LIN {X 0,Y 573.243,Z 513.073,A -85,B 0,C 180,E1 -2300.392,E2 -2300.392} C_VEL
LIN {X 0,Y 573.249,Z 513.077,A -85,B 0,C 180,E1 -2303.077,E2 -2303.077} C_VEL
LIN {X 0,Y 573.268,Z 513.077,A -85,B 0,C 180,E1 -2305.671,E2 -2305.671} C_VEL
LIN {X 0,Y 573.242,Z 513.074,A -85,B 0,C 180,E1 -2308.184,E2 -2308.184} C_VEL
LIN {X 0,Y 573.262,Z 513.071,A -85,B 0,C 180,E1 -2310.634,E2 -2310.634} C_VEL
LIN {X 0,Y 573.262,Z 513.081,A -85,B 0,C 180,E1 -2313.499,E2 -2313.499} C_VEL
LIN {X 0,Y 573.224,Z 513.076,A -85,B 0,C 180,E1 -2316.134,E2 -2316.134} C_VEL
LIN {X 0,Y 573.253,Z 513.078,A -85,B 0,C 180,E1 -2319.173,E2 -2319.173} C_VEL
LIN {X 0,Y 573.231,Z 513.084,A -85,B 0,C 180,E1 -2321.411,E2 -2321.411} C_VEL
LIN {X 0,Y 573.249,Z 513.079,A -85,B 0,C 180,E1 -2323.621,E2 -2323.621} C_VEL
LIN {X 0,Y 573.227,Z 513.076,A -85,B 0,C 180,E1 -2326.529,E2 -2326.529} C_VEL
LIN {X 0,Y 573.273,Z 513.07,A -85,B 0,C 180,E1 -2328.733,E2 -2328.733} C_VEL
LIN {X 0,Y 573.298,Z 513.075,A -85,B 0,C 180,E1 -2331.54,E2 -2331.54} C_VEL
LIN {X 0,Y 573.284,Z 513.068,A -85,B 0,C 180,E1 -2334.371,E2 -2334.371} C_VEL
LIN {X 0,Y 573.3,Z 513.069,A -85,B 0,C 180,E1 -2337.892,E2 -2337.892} C_VEL
LIN {X 0,Y 573.328,Z 513.064,A -85,B 0,C 180,E1 -2340.702,E2 -2340.702} C_VEL
LIN {X 0,Y 573.234,Z 513.083,A -85,B 0,C 180,E1 -2343.514,E2 -2343.514} C_VEL
LIN {X 0,Y 573.283,Z 513.075,A -85,B 0,C 180,E1 -2345.628,E2 -2345.628} C_VEL
LIN {X 0,Y 573.298,Z 513.067,A -85,B 0,C 180,E1 -2348.459,E2 -2348.459} C_VEL
LIN {X 0,Y 573.287,Z 513.077,A -85,B 0,C 180,E1 -2351.311,E2 -2351.311} C_VEL
LIN {X 0,Y 573.269,Z 513.071,A -85,B 0,C 180,E1 -2354.425,E2 -2354.425} C_VEL
LIN {X 0,Y 573.249,Z 513.079,A -85,B 0,C 180,E1 -2357.111,E2 -2357.111} C_VEL
LIN {X 0,Y 573.247,Z 513.075,A -85,B 0,C 180,E1 -2360.076,E2 -2360.076} C_VEL
LIN {X 0,Y 573.229,Z 513.076,A -85,B 0,C 180,E1 -2362.338,E2 -2362.338} C_VEL
LIN {X 0,Y 573.24,Z 513.075,A -85,B 0,C 180,E1 -2364.401,E2 -2364.401} C_VEL
LIN {X 0,Y 572.615,Z 513.157,A -85,B 0,C 180,E1 -2364.987,E2 -2364.987} C_VEL
LIN {X 0,Y 569.777,Z 513.516,A -85,B 0,C 180,E1 -2365.939,E2 -2365.939} C_VEL
LIN {X 0,Y 567.349,Z 513.821,A -85,B 0,C 180,E1 -2366.705,E2 -2366.705} C_VEL
LIN {X 0,Y 566.296,Z 513.949,A -85,B 0,C 180,E1 -2367.296,E2 -2367.296} C_VEL
LIN {X 0,Y 566.207,Z 513.958,A -85,B 0,C 180,E1 -2367.496,E2 -2367.496} C_VEL
LIN {X 0,Y 566.246,Z 514.057,A -85,B 0,C 180,E1 -2370.176,E2 -2370.176} C_VEL
LIN {X 0,Y 566.585,Z 517.753,A -85,B 0,C 180,E1 -2370.853,E2 -2370.853} C_VEL
LIN {X 0,Y 566.382,Z 534.137,A -85,B 0,C 180,E1 -2373.762,E2 -2373.762} C_VEL
LIN {X 0,Y 566.229,Z 547.137,A -85,B 0,C 180,E1 -2376.042,E2 -2376.042} C_VEL
LIN {X 0,Y 567.189,Z 554.187,A -85,B 0,C 180,E1 -2376.165,E2 -2376.165} C_VEL
LIN {X 0,Y 566.935,Z 654.262,A -85,B 0,C 180,E1 -2377.453,E2 -2377.453} C_VEL
LIN {X 0,Y 566.822,Z 667.928,A -85,B 0,C 180,E1 -2377.785,E2 -2377.785} C_VEL
LIN {X 0,Y 566.718,Z 679.77,A -85,B 0,C 180,E1 -2378.209,E2 -2378.209} C_VEL
LIN {X 0,Y 566.6,Z 691.935,A -85,B 0,C 180,E1 -2378.797,E2 -2378.797} C_VEL
LIN {X 0,Y 566.436,Z 702.934,A -85,B 0,C 180,E1 -2379.48,E2 -2379.48} C_VEL
LIN {X 0,Y 566.311,Z 713.502,A -85,B 0,C 180,E1 -2380.301,E2 -2380.301} C_VEL
LIN {X 0,Y 566.196,Z 723.392,A -85,B 0,C 180,E1 -2381.255,E2 -2381.255} C_VEL
LIN {X 0,Y 566.063,Z 732.117,A -85,B 0,C 180,E1 -2382.297,E2 -2382.297} C_VEL
LIN {X 0,Y 565.987,Z 738.863,A -85,B 0,C 180,E1 -2383.288,E2 -2383.288} C_VEL
LIN {X 0,Y 565.955,Z 745.455,A -85,B 0,C 180,E1 -2384.502,E2 -2384.502} C_VEL
LIN {X 0,Y 565.911,Z 749.683,A -85,B 0,C 180,E1 -2385.495,E2 -2385.495} C_VEL
LIN {X 0,Y 565.888,Z 753.006,A -85,B 0,C 180,E1 -2386.5,E2 -2386.5} C_VEL
LIN {X 0,Y 565.861,Z 756.162,A -85,B 0,C 180,E1 -2387.882,E2 -2387.882} C_VEL
LIN {X 0,Y 565.825,Z 757.735,A -85,B 0,C 180,E1 -2389.258,E2 -2389.258} C_VEL
LIN {X 0,Y 565.812,Z 757.824,A -85,B 0,C 180,E1 -2390.695,E2 -2390.695} C_VEL
LIN {X 0,Y 565.827,Z 757.03,A -85,B 0,C 180,E1 -2391.61,E2 -2391.61} C_VEL
LIN {X 0,Y 565.843,Z 755.324,A -85,B 0,C 180,E1 -2392.646,E2 -2392.646} C_VEL
LIN {X 0,Y 565.912,Z 752.312,A -85,B 0,C 180,E1 -2393.825,E2 -2393.825} C_VEL
LIN {X 0,Y 565.9,Z 747.388,A -85,B 0,C 180,E1 -2395.162,E2 -2395.162} C_VEL
LIN {X 0,Y 565.984,Z 741.795,A -85,B 0,C 180,E1 -2396.3,E2 -2396.3} C_VEL
LIN {X 0,Y 566.048,Z 734.523,A -85,B 0,C 180,E1 -2397.462,E2 -2397.462} C_VEL
LIN {X 0,Y 566.173,Z 725.725,A -85,B 0,C 180,E1 -2398.578,E2 -2398.578} C_VEL
LIN {X 0,Y 566.257,Z 716.551,A -85,B 0,C 180,E1 -2399.516,E2 -2399.516} C_VEL
LIN {X 0,Y 566.398,Z 706.371,A -85,B 0,C 180,E1 -2400.362,E2 -2400.362} C_VEL
LIN {X 0,Y 566.515,Z 695.904,A -85,B 0,C 180,E1 -2401.066,E2 -2401.066} C_VEL
LIN {X 0,Y 566.678,Z 683.715,A -85,B 0,C 180,E1 -2401.708,E2 -2401.708} C_VEL
LIN {X 0,Y 566.802,Z 671.491,A -85,B 0,C 180,E1 -2402.192,E2 -2402.192} C_VEL
LIN {X 0,Y 566.923,Z 658.595,A -85,B 0,C 180,E1 -2402.549,E2 -2402.549} C_VEL
LIN {X 0,Y 567.017,Z 643.292,A -85,B 0,C 180,E1 -2402.793,E2 -2402.793} C_VEL
LIN {X 0,Y 567.092,Z 552.392,A -85,B 0,C 180,E1 -2403.95,E2 -2403.95} C_VEL
LIN {X 0,Y 566.244,Z 547.089,A -85,B 0,C 180,E1 -2404.056,E2 -2404.056} C_VEL
LIN {X 0,Y 566.406,Z 531.183,A -85,B 0,C 180,E1 -2406.849,E2 -2406.849} C_VEL
LIN {X 0,Y 566.53,Z 516.374,A -85,B 0,C 180,E1 -2409.486,E2 -2409.486} C_VEL
LIN {X 0,Y 566.234,Z 513.954,A -85,B 0,C 180,E1 -2409.949,E2 -2409.949} C_VEL
LIN {X 0,Y 566.22,Z 513.957,A -85,B 0,C 180,E1 -2412.887,E2 -2412.887} C_VEL
LIN {X 0,Y 566.23,Z 513.948,A -85,B 0,C 180,E1 -2415.628,E2 -2415.628} C_VEL
LIN {X 0,Y 566.23,Z 513.955,A -85,B 0,C 180,E1 -2418.676,E2 -2418.676} C_VEL
LIN {X 0,Y 566.226,Z 513.949,A -85,B 0,C 180,E1 -2421.435,E2 -2421.435} C_VEL
LIN {X 0,Y 566.263,Z 513.945,A -85,B 0,C 180,E1 -2424.303,E2 -2424.303} C_VEL
LIN {X 0,Y 566.282,Z 513.94,A -85,B 0,C 180,E1 -2427.867,E2 -2427.867} C_VEL
LIN {X 0,Y 566.301,Z 513.944,A -85,B 0,C 180,E1 -2430.712,E2 -2430.712} C_VEL
LIN {X 0,Y 566.27,Z 513.95,A -85,B 0,C 180,E1 -2432.847,E2 -2432.847} C_VEL
LIN {X 0,Y 566.261,Z 513.944,A -85,B 0,C 180,E1 -2435.699,E2 -2435.699} C_VEL
LIN {X 0,Y 566.226,Z 513.951,A -85,B 0,C 180,E1 -2438.567,E2 -2438.567} C_VEL
LIN {X 0,Y 566.241,Z 513.949,A -85,B 0,C 180,E1 -2441.455,E2 -2441.455} C_VEL
LIN {X 0,Y 566.234,Z 513.948,A -85,B 0,C 180,E1 -2444.508,E2 -2444.508} C_VEL
LIN {X 0,Y 566.199,Z 513.957,A -85,B 0,C 180,E1 -2447.333,E2 -2447.333} C_VEL
LIN {X 0,Y 566.213,Z 513.949,A -85,B 0,C 180,E1 -2450.338,E2 -2450.338} C_VEL
LIN {X 0,Y 566.17,Z 513.962,A -85,B 0,C 180,E1 -2453.282,E2 -2453.282} C_VEL
LIN {X 0,Y 566.213,Z 513.951,A -85,B 0,C 180,E1 -2455.75,E2 -2455.75} C_VEL
LIN {X 0,Y 566.203,Z 513.95,A -85,B 0,C 180,E1 -2458.203,E2 -2458.203} C_VEL
LIN {X 0,Y 566.201,Z 513.958,A -85,B 0,C 180,E1 -2461.079,E2 -2461.079} C_VEL
LIN {X 0,Y 566.213,Z 513.952,A -85,B 0,C 180,E1 -2463.735,E2 -2463.735} C_VEL
LIN {X 0,Y 566.201,Z 513.951,A -85,B 0,C 180,E1 -2466.571,E2 -2466.571} C_VEL
LIN {X 0,Y 566.223,Z 513.958,A -85,B 0,C 180,E1 -2469.274,E2 -2469.274} C_VEL
LIN {X 0,Y 566.217,Z 513.949,A -85,B 0,C 180,E1 -2472.088,E2 -2472.088} C_VEL
LIN {X 0,Y 566.176,Z 513.958,A -85,B 0,C 180,E1 -2475.037,E2 -2475.037} C_VEL
LIN {X 0,Y 566.191,Z 513.954,A -85,B 0,C 180,E1 -2477.911,E2 -2477.911} C_VEL
LIN {X 0,Y 566.224,Z 513.948,A -85,B 0,C 180,E1 -2480.728,E2 -2480.728} C_VEL
LIN {X 0,Y 566.188,Z 513.957,A -85,B 0,C 180,E1 -2483.789,E2 -2483.789} C_VEL
LIN {X 0,Y 566.216,Z 513.949,A -85,B 0,C 180,E1 -2486.266,E2 -2486.266} C_VEL
LIN {X 0,Y 566.194,Z 513.953,A -85,B 0,C 180,E1 -2488.924,E2 -2488.924} C_VEL
LIN {X 0,Y 566.216,Z 513.954,A -85,B 0,C 180,E1 -2491.858,E2 -2491.858} C_VEL
LIN {X 0,Y 566.219,Z 513.949,A -85,B 0,C 180,E1 -2494.252,E2 -2494.252} C_VEL
LIN {X 0,Y 566.174,Z 513.954,A -85,B 0,C 180,E1 -2496.72,E2 -2496.72} C_VEL
LIN {X 0,Y 566.212,Z 513.959,A -85,B 0,C 180,E1 -2499.663,E2 -2499.663} C_VEL
LIN {X 0,Y 566.205,Z 513.95,A -85,B 0,C 180,E1 -2502.669,E2 -2502.669} C_VEL
LIN {X 0,Y 566.239,Z 513.955,A -85,B 0,C 180,E1 -2505.627,E2 -2505.627} C_VEL
LIN {X 0,Y 566.241,Z 513.945,A -85,B 0,C 180,E1 -2508.676,E2 -2508.676} C_VEL
LIN {X 0,Y 566.233,Z 513.952,A -85,B 0,C 180,E1 -2511.435,E2 -2511.435} C_VEL
LIN {X 0,Y 566.261,Z 513.945,A -85,B 0,C 180,E1 -2514.302,E2 -2514.302} C_VEL
LIN {X 0,Y 566.285,Z 513.949,A -85,B 0,C 180,E1 -2517.867,E2 -2517.867} C_VEL
LIN {X 0,Y 566.307,Z 513.937,A -85,B 0,C 180,E1 -2520.711,E2 -2520.711} C_VEL
LIN {X 0,Y 566.278,Z 513.941,A -85,B 0,C 180,E1 -2522.846,E2 -2522.846} C_VEL
LIN {X 0,Y 566.264,Z 513.95,A -85,B 0,C 180,E1 -2525.699,E2 -2525.699} C_VEL
LIN {X 0,Y 566.233,Z 513.948,A -85,B 0,C 180,E1 -2528.566,E2 -2528.566} C_VEL
LIN {X 0,Y 566.249,Z 513.947,A -85,B 0,C 180,E1 -2531.455,E2 -2531.455} C_VEL
LIN {X 0,Y 566.242,Z 513.948,A -85,B 0,C 180,E1 -2534.507,E2 -2534.507} C_VEL
LIN {X 0,Y 566.206,Z 513.951,A -85,B 0,C 180,E1 -2537.332,E2 -2537.332} C_VEL
LIN {X 0,Y 566.215,Z 513.954,A -85,B 0,C 180,E1 -2540.337,E2 -2540.337} C_VEL
LIN {X 0,Y 566.177,Z 513.954,A -85,B 0,C 180,E1 -2543.281,E2 -2543.281} C_VEL
LIN {X 0,Y 566.22,Z 513.953,A -85,B 0,C 180,E1 -2545.749,E2 -2545.749} C_VEL
LIN {X 0,Y 566.21,Z 513.958,A -85,B 0,C 180,E1 -2548.202,E2 -2548.202} C_VEL
LIN {X 0,Y 566.197,Z 513.951,A -85,B 0,C 180,E1 -2551.076,E2 -2551.076} C_VEL
LIN {X 0,Y 566.205,Z 513.953,A -85,B 0,C 180,E1 -2553.732,E2 -2553.732} C_VEL
LIN {X 0,Y 566.215,Z 513.953,A -85,B 0,C 180,E1 -2556.569,E2 -2556.569} C_VEL
LIN {X 0,Y 566.222,Z 513.95,A -85,B 0,C 180,E1 -2559.686,E2 -2559.686} C_VEL
LIN {X 0,Y 566.2,Z 513.952,A -85,B 0,C 180,E1 -2562.916,E2 -2562.916} C_VEL
LIN {X 0,Y 566.206,Z 513.956,A -85,B 0,C 180,E1 -2566.048,E2 -2566.048} C_VEL
LIN {X 0,Y 566.211,Z 513.949,A -85,B 0,C 180,E1 -2569.214,E2 -2569.214} C_VEL
LIN {X 0,Y 566.19,Z 513.953,A -85,B 0,C 180,E1 -2571.636,E2 -2571.636} C_VEL
LIN {X 0,Y 566.169,Z 513.964,A -85,B 0,C 180,E1 -2574.307,E2 -2574.307} C_VEL
LIN {X 0,Y 566.227,Z 513.95,A -85,B 0,C 180,E1 -2576.897,E2 -2576.897} C_VEL
LIN {X 0,Y 566.187,Z 513.953,A -85,B 0,C 180,E1 -2579.407,E2 -2579.407} C_VEL
LIN {X 0,Y 566.219,Z 513.95,A -85,B 0,C 180,E1 -2581.857,E2 -2581.857} C_VEL
LIN {X 0,Y 566.216,Z 513.956,A -85,B 0,C 180,E1 -2584.25,E2 -2584.25} C_VEL
LIN {X 0,Y 566.187,Z 514.013,A -85,B 0,C 180,E1 -2586.754,E2 -2586.754} C_VEL
LIN {X 0,Y 567.076,Z 519.274,A -85,B 0,C 180,E1 -2587.597,E2 -2587.597} C_VEL
LIN {X 0,Y 566.791,Z 539.041,A -85,B 0,C 180,E1 -2590.571,E2 -2590.571} C_VEL
LIN {X 0,Y 566.558,Z 557.196,A -85,B 0,C 180,E1 -2593.257,E2 -2593.257} C_VEL
LIN {X 0,Y 566.399,Z 576.069,A -85,B 0,C 180,E1 -2595.997,E2 -2595.997} C_VEL
LIN {X 0,Y 567.211,Z 583.224,A -85,B 0,C 180,E1 -2596.109,E2 -2596.109} C_VEL
LIN {X 0,Y 566.94,Z 683.899,A -85,B 0,C 180,E1 -2597.402,E2 -2597.402} C_VEL
LIN {X 0,Y 566.837,Z 697.187,A -85,B 0,C 180,E1 -2597.718,E2 -2597.718} C_VEL
LIN {X 0,Y 566.758,Z 709.351,A -85,B 0,C 180,E1 -2598.148,E2 -2598.148} C_VEL
LIN {X 0,Y 566.606,Z 721.341,A -85,B 0,C 180,E1 -2598.718,E2 -2598.718} C_VEL
LIN {X 0,Y 566.461,Z 733.188,A -85,B 0,C 180,E1 -2599.454,E2 -2599.454} C_VEL
LIN {X 0,Y 566.319,Z 743.59,A -85,B 0,C 180,E1 -2600.264,E2 -2600.264} C_VEL
LIN {X 0,Y 566.207,Z 752.103,A -85,B 0,C 180,E1 -2601.073,E2 -2601.073} C_VEL
LIN {X 0,Y 566.113,Z 759.953,A -85,B 0,C 180,E1 -2601.971,E2 -2601.971} C_VEL
LIN {X 0,Y 566.005,Z 767.615,A -85,B 0,C 180,E1 -2603.046,E2 -2603.046} C_VEL
LIN {X 0,Y 566.004,Z 774.675,A -85,B 0,C 180,E1 -2604.298,E2 -2604.298} C_VEL
LIN {X 0,Y 565.933,Z 779.368,A -85,B 0,C 180,E1 -2605.369,E2 -2605.369} C_VEL
LIN {X 0,Y 565.927,Z 782.954,A -85,B 0,C 180,E1 -2606.439,E2 -2606.439} C_VEL
LIN {X 0,Y 565.878,Z 784.806,A -85,B 0,C 180,E1 -2607.151,E2 -2607.151} C_VEL
LIN {X 0,Y 565.846,Z 787.185,A -85,B 0,C 180,E1 -2608.576,E2 -2608.576} C_VEL
LIN {X 0,Y 565.839,Z 788,A -85,B 0,C 180,E1 -2609.999,E2 -2609.999} C_VEL
LIN {X 0,Y 565.846,Z 787.188,A -85,B 0,C 180,E1 -2611.422,E2 -2611.422} C_VEL
LIN {X 0,Y 565.878,Z 784.812,A -85,B 0,C 180,E1 -2612.847,E2 -2612.847} C_VEL
LIN {X 0,Y 565.926,Z 781.899,A -85,B 0,C 180,E1 -2613.915,E2 -2613.915} C_VEL
LIN {X 0,Y 565.878,Z 777.953,A -85,B 0,C 180,E1 -2614.986,E2 -2614.986} C_VEL
LIN {X 0,Y 566.001,Z 772.872,A -85,B 0,C 180,E1 -2616.057,E2 -2616.057} C_VEL
LIN {X 0,Y 566.04,Z 766.476,A -85,B 0,C 180,E1 -2617.131,E2 -2617.131} C_VEL
LIN {X 0,Y 566.133,Z 758.487,A -85,B 0,C 180,E1 -2618.207,E2 -2618.207} C_VEL
LIN {X 0,Y 566.228,Z 750.347,A -85,B 0,C 180,E1 -2619.104,E2 -2619.104} C_VEL
LIN {X 0,Y 566.34,Z 740.414,A -85,B 0,C 180,E1 -2620.004,E2 -2620.004} C_VEL
LIN {X 0,Y 566.514,Z 729.301,A -85,B 0,C 180,E1 -2620.807,E2 -2620.807} C_VEL
LIN {X 0,Y 566.659,Z 718.199,A -85,B 0,C 180,E1 -2621.445,E2 -2621.445} C_VEL
LIN {X 0,Y 566.738,Z 706.012,A -85,B 0,C 180,E1 -2621.987,E2 -2621.987} C_VEL
LIN {X 0,Y 566.911,Z 693.222,A -85,B 0,C 180,E1 -2622.392,E2 -2622.392} C_VEL
LIN {X 0,Y 566.981,Z 681.182,A -85,B 0,C 180,E1 -2622.641,E2 -2622.641} C_VEL
LIN {X 0,Y 567.029,Z 580.268,A -85,B 0,C 180,E1 -2623.934,E2 -2623.934} C_VEL
LIN {X 0,Y 566.389,Z 575.8,A -85,B 0,C 180,E1 -2624.024,E2 -2624.024} C_VEL
LIN {X 0,Y 566.587,Z 554.721,A -85,B 0,C 180,E1 -2627.107,E2 -2627.107} C_VEL
LIN {X 0,Y 566.849,Z 534.4,A -85,B 0,C 180,E1 -2630.123,E2 -2630.123} C_VEL
LIN {X 0,Y 567.093,Z 519.288,A -85,B 0,C 180,E1 -2632.4,E2 -2632.4} C_VEL
LIN {X 0,Y 566.188,Z 513.964,A -85,B 0,C 180,E1 -2633.284,E2 -2633.284} C_VEL
LIN {X 0,Y 566.212,Z 513.957,A -85,B 0,C 180,E1 -2635.748,E2 -2635.748} C_VEL
LIN {X 0,Y 566.2,Z 513.954,A -85,B 0,C 180,E1 -2638.201,E2 -2638.201} C_VEL
LIN {X 0,Y 566.197,Z 513.957,A -85,B 0,C 180,E1 -2641.077,E2 -2641.077} C_VEL
LIN {X 0,Y 566.208,Z 513.956,A -85,B 0,C 180,E1 -2643.733,E2 -2643.733} C_VEL
LIN {X 0,Y 566.207,Z 513.951,A -85,B 0,C 180,E1 -2646.568,E2 -2646.568} C_VEL
LIN {X 0,Y 566.208,Z 513.957,A -85,B 0,C 180,E1 -2649.684,E2 -2649.684} C_VEL
LIN {X 0,Y 566.21,Z 513.952,A -85,B 0,C 180,E1 -2652.086,E2 -2652.086} C_VEL
LIN {X 0,Y 566.167,Z 513.959,A -85,B 0,C 180,E1 -2655.035,E2 -2655.035} C_VEL
LIN {X 0,Y 566.211,Z 513.951,A -85,B 0,C 180,E1 -2658.135,E2 -2658.135} C_VEL
LIN {X 0,Y 566.216,Z 513.95,A -85,B 0,C 180,E1 -2660.726,E2 -2660.726} C_VEL
LIN {X 0,Y 566.211,Z 513.954,A -85,B 0,C 180,E1 -2663.782,E2 -2663.782} C_VEL
LIN {X 0,Y 566.222,Z 513.948,A -85,B 0,C 180,E1 -2666.262,E2 -2666.262} C_VEL
LIN {X 0,Y 566.194,Z 513.954,A -85,B 0,C 180,E1 -2668.92,E2 -2668.92} C_VEL
LIN {X 0,Y 566.189,Z 513.956,A -85,B 0,C 180,E1 -2671.046,E2 -2671.046} C_VEL
LIN {X 0,Y 566.237,Z 513.956,A -85,B 0,C 180,E1 -2673.46,E2 -2673.46} C_VEL
LIN {X 0,Y 566.19,Z 513.955,A -85,B 0,C 180,E1 -2675.819,E2 -2675.819} C_VEL
LIN {X 0,Y 566.208,Z 513.952,A -85,B 0,C 180,E1 -2678.902,E2 -2678.902} C_VEL
LIN {X 0,Y 566.205,Z 513.955,A -85,B 0,C 180,E1 -2681.172,E2 -2681.172} C_VEL
LIN {X 0,Y 566.211,Z 513.959,A -85,B 0,C 180,E1 -2683.412,E2 -2683.412} C_VEL
LIN {X 0,Y 566.19,Z 513.952,A -85,B 0,C 180,E1 -2686.358,E2 -2686.358} C_VEL
LIN {X 0,Y 566.265,Z 513.942,A -85,B 0,C 180,E1 -2688.653,E2 -2688.653} C_VEL
LIN {X 0,Y 566.239,Z 513.955,A -85,B 0,C 180,E1 -2691.434,E2 -2691.434} C_VEL
LIN {X 0,Y 566.251,Z 513.945,A -85,B 0,C 180,E1 -2694.301,E2 -2694.301} C_VEL
LIN {X 0,Y 566.271,Z 513.945,A -85,B 0,C 180,E1 -2697.866,E2 -2697.866} C_VEL
LIN {X 0,Y 566.298,Z 513.94,A -85,B 0,C 180,E1 -2700.711,E2 -2700.711} C_VEL
LIN {X 0,Y 566.27,Z 513.944,A -85,B 0,C 180,E1 -2702.845,E2 -2702.845} C_VEL
LIN {X 0,Y 566.251,Z 513.95,A -85,B 0,C 180,E1 -2705.698,E2 -2705.698} C_VEL
LIN {X 0,Y 566.239,Z 513.947,A -85,B 0,C 180,E1 -2708.565,E2 -2708.565} C_VEL
LIN {X 0,Y 566.239,Z 513.956,A -85,B 0,C 180,E1 -2711.454,E2 -2711.454} C_VEL
LIN {X 0,Y 566.222,Z 513.949,A -85,B 0,C 180,E1 -2714.507,E2 -2714.507} C_VEL
LIN {X 0,Y 566.194,Z 513.962,A -85,B 0,C 180,E1 -2717.331,E2 -2717.331} C_VEL
LIN {X 0,Y 566.209,Z 513.95,A -85,B 0,C 180,E1 -2720.337,E2 -2720.337} C_VEL
LIN {X 0,Y 566.179,Z 513.963,A -85,B 0,C 180,E1 -2723.404,E2 -2723.404} C_VEL
LIN {X 0,Y 566.216,Z 513.955,A -85,B 0,C 180,E1 -2725.748,E2 -2725.748} C_VEL
LIN {X 0,Y 566.207,Z 513.958,A -85,B 0,C 180,E1 -2727.496,E2 -2727.496} C_VEL
LIN {X 0,Y 565.52,Z 514.041,A -85,B 0,C 180,E1 -2727.892,E2 -2727.892} C_VEL
LIN {X 0,Y 559.819,Z 514.755,A -85,B 0,C 180,E1 -2729.137,E2 -2729.137} C_VEL
LIN {X 0,Y 559.155,Z 514.837,A -85,B 0,C 180,E1 -2729.54,E2 -2729.54} C_VEL
LIN {X 0,Y 559.213,Z 514.972,A -85,B 0,C 180,E1 -2730.083,E2 -2730.083} C_VEL
LIN {X 0,Y 559.566,Z 519.903,A -85,B 0,C 180,E1 -2730.994,E2 -2730.994} C_VEL
LIN {X 0,Y 559.377,Z 535.33,A -85,B 0,C 180,E1 -2733.766,E2 -2733.766} C_VEL
LIN {X 0,Y 559.188,Z 547.236,A -85,B 0,C 180,E1 -2735.873,E2 -2735.873} C_VEL
LIN {X 0,Y 560.272,Z 553.876,A -85,B 0,C 180,E1 -2735.987,E2 -2735.987} C_VEL
LIN {X 0,Y 560.022,Z 654.191,A -85,B 0,C 180,E1 -2737.293,E2 -2737.293} C_VEL
LIN {X 0,Y 559.9,Z 667.815,A -85,B 0,C 180,E1 -2737.627,E2 -2737.627} C_VEL
LIN {X 0,Y 559.755,Z 680.312,A -85,B 0,C 180,E1 -2738.081,E2 -2738.081} C_VEL
LIN {X 0,Y 559.621,Z 692.123,A -85,B 0,C 180,E1 -2738.666,E2 -2738.666} C_VEL
LIN {X 0,Y 559.433,Z 703.358,A -85,B 0,C 180,E1 -2739.376,E2 -2739.376} C_VEL
LIN {X 0,Y 559.296,Z 714.193,A -85,B 0,C 180,E1 -2740.239,E2 -2740.239} C_VEL
LIN {X 0,Y 559.136,Z 723.82,A -85,B 0,C 180,E1 -2741.19,E2 -2741.19} C_VEL
LIN {X 0,Y 559.007,Z 732.434,A -85,B 0,C 180,E1 -2742.241,E2 -2742.241} C_VEL
LIN {X 0,Y 558.896,Z 740.27,A -85,B 0,C 180,E1 -2743.44,E2 -2743.44} C_VEL
LIN {X 0,Y 558.863,Z 745.614,A -85,B 0,C 180,E1 -2744.465,E2 -2744.465} C_VEL
LIN {X 0,Y 558.814,Z 750.957,A -85,B 0,C 180,E1 -2745.796,E2 -2745.796} C_VEL
LIN {X 0,Y 558.759,Z 754.941,A -85,B 0,C 180,E1 -2747.22,E2 -2747.22} C_VEL
LIN {X 0,Y 558.756,Z 756.676,A -85,B 0,C 180,E1 -2748.194,E2 -2748.194} C_VEL
LIN {X 0,Y 558.742,Z 757.674,A -85,B 0,C 180,E1 -2749.153,E2 -2749.153} C_VEL
LIN {X 0,Y 558.753,Z 757.993,A -85,B 0,C 180,E1 -2750.108,E2 -2750.108} C_VEL
LIN {X 0,Y 558.724,Z 757.44,A -85,B 0,C 180,E1 -2751.249,E2 -2751.249} C_VEL
LIN {X 0,Y 558.744,Z 755.844,A -85,B 0,C 180,E1 -2752.412,E2 -2752.412} C_VEL
LIN {X 0,Y 558.835,Z 752.621,A -85,B 0,C 180,E1 -2753.768,E2 -2753.768} C_VEL
LIN {X 0,Y 558.804,Z 748.993,A -85,B 0,C 180,E1 -2754.834,E2 -2754.834} C_VEL
LIN {X 0,Y 558.871,Z 743.311,A -85,B 0,C 180,E1 -2756.095,E2 -2756.095} C_VEL
LIN {X 0,Y 558.948,Z 736.432,A -85,B 0,C 180,E1 -2757.273,E2 -2757.273} C_VEL
LIN {X 0,Y 559.049,Z 729.01,A -85,B 0,C 180,E1 -2758.295,E2 -2758.295} C_VEL
LIN {X 0,Y 559.193,Z 720.027,A -85,B 0,C 180,E1 -2759.299,E2 -2759.299} C_VEL
LIN {X 0,Y 559.329,Z 710.35,A -85,B 0,C 180,E1 -2760.179,E2 -2760.179} C_VEL
LIN {X 0,Y 559.475,Z 699.524,A -85,B 0,C 180,E1 -2760.976,E2 -2760.976} C_VEL
LIN {X 0,Y 559.644,Z 688.739,A -85,B 0,C 180,E1 -2761.608,E2 -2761.608} C_VEL
LIN {X 0,Y 559.827,Z 676.28,A -85,B 0,C 180,E1 -2762.172,E2 -2762.172} C_VEL
LIN {X 0,Y 559.943,Z 663.4,A -85,B 0,C 180,E1 -2762.589,E2 -2762.589} C_VEL
LIN {X 0,Y 560.047,Z 650.613,A -85,B 0,C 180,E1 -2762.853,E2 -2762.853} C_VEL
LIN {X 0,Y 560.246,Z 553.607,A -85,B 0,C 180,E1 -2764.108,E2 -2764.108} C_VEL
LIN {X 0,Y 559.228,Z 547.111,A -85,B 0,C 180,E1 -2764.232,E2 -2764.232} C_VEL
LIN {X 0,Y 559.468,Z 529.99,A -85,B 0,C 180,E1 -2767.278,E2 -2767.278} C_VEL
LIN {X 0,Y 559.506,Z 517.138,A -85,B 0,C 180,E1 -2769.601,E2 -2769.601} C_VEL
LIN {X 0,Y 559.197,Z 514.831,A -85,B 0,C 180,E1 -2770.069,E2 -2770.069} C_VEL
LIN {X 0,Y 559.178,Z 514.83,A -85,B 0,C 180,E1 -2773.199,E2 -2773.199} C_VEL
LIN {X 0,Y 559.171,Z 514.829,A -85,B 0,C 180,E1 -2776.185,E2 -2776.185} C_VEL
LIN {X 0,Y 559.191,Z 514.828,A -85,B 0,C 180,E1 -2779.135,E2 -2779.135} C_VEL
LIN {X 0,Y 559.203,Z 514.823,A -85,B 0,C 180,E1 -2782.055,E2 -2782.055} C_VEL
LIN {X 0,Y 559.252,Z 514.825,A -85,B 0,C 180,E1 -2784.954,E2 -2784.954} C_VEL
LIN {X 0,Y 559.253,Z 514.816,A -85,B 0,C 180,E1 -2787.84,E2 -2787.84} C_VEL
LIN {X 0,Y 559.271,Z 514.82,A -85,B 0,C 180,E1 -2790.721,E2 -2790.721} C_VEL
LIN {X 0,Y 559.237,Z 514.827,A -85,B 0,C 180,E1 -2792.882,E2 -2792.882} C_VEL
LIN {X 0,Y 559.229,Z 514.819,A -85,B 0,C 180,E1 -2795.771,E2 -2795.771} C_VEL
LIN {X 0,Y 559.185,Z 514.829,A -85,B 0,C 180,E1 -2798.675,E2 -2798.675} C_VEL
LIN {X 0,Y 559.205,Z 514.824,A -85,B 0,C 180,E1 -2801.601,E2 -2801.601} C_VEL
LIN {X 0,Y 559.199,Z 514.825,A -85,B 0,C 180,E1 -2804.596,E2 -2804.596} C_VEL
LIN {X 0,Y 559.142,Z 514.833,A -85,B 0,C 180,E1 -2807.558,E2 -2807.558} C_VEL
LIN {X 0,Y 559.172,Z 514.827,A -85,B 0,C 180,E1 -2809.838,E2 -2809.838} C_VEL
LIN {X 0,Y 559.141,Z 514.83,A -85,B 0,C 180,E1 -2812.154,E2 -2812.154} C_VEL
LIN {X 0,Y 559.176,Z 514.834,A -85,B 0,C 180,E1 -2815.299,E2 -2815.299} C_VEL
LIN {X 0,Y 559.158,Z 514.83,A -85,B 0,C 180,E1 -2817.714,E2 -2817.714} C_VEL
LIN {X 0,Y 559.158,Z 514.828,A -85,B 0,C 180,E1 -2820.183,E2 -2820.183} C_VEL
LIN {X 0,Y 559.159,Z 514.83,A -85,B 0,C 180,E1 -2822.716,E2 -2822.716} C_VEL
LIN {X 0,Y 559.129,Z 514.841,A -85,B 0,C 180,E1 -2825.325,E2 -2825.325} C_VEL
LIN {X 0,Y 559.137,Z 514.831,A -85,B 0,C 180,E1 -2828.018,E2 -2828.018} C_VEL
LIN {X 0,Y 559.193,Z 514.829,A -85,B 0,C 180,E1 -2831.055,E2 -2831.055} C_VEL
LIN {X 0,Y 559.165,Z 514.831,A -85,B 0,C 180,E1 -2833.732,E2 -2833.732} C_VEL
LIN {X 0,Y 559.148,Z 514.831,A -85,B 0,C 180,E1 -2836.804,E2 -2836.804} C_VEL
LIN {X 0,Y 559.176,Z 514.832,A -85,B 0,C 180,E1 -2839.19,E2 -2839.19} C_VEL
LIN {X 0,Y 559.137,Z 514.833,A -85,B 0,C 180,E1 -2841.983,E2 -2841.983} C_VEL
LIN {X 0,Y 559.138,Z 514.831,A -85,B 0,C 180,E1 -2844.787,E2 -2844.787} C_VEL
LIN {X 0,Y 559.177,Z 514.833,A -85,B 0,C 180,E1 -2847.362,E2 -2847.362} C_VEL
LIN {X 0,Y 559.153,Z 514.83,A -85,B 0,C 180,E1 -2850.143,E2 -2850.143} C_VEL
LIN {X 0,Y 559.173,Z 514.829,A -85,B 0,C 180,E1 -2853.098,E2 -2853.098} C_VEL
LIN {X 0,Y 559.161,Z 514.836,A -85,B 0,C 180,E1 -2855.496,E2 -2855.496} C_VEL
LIN {X 0,Y 559.177,Z 514.825,A -85,B 0,C 180,E1 -2858.625,E2 -2858.625} C_VEL
LIN {X 0,Y 559.167,Z 514.827,A -85,B 0,C 180,E1 -2860.927,E2 -2860.927} C_VEL
LIN {X 0,Y 559.171,Z 514.832,A -85,B 0,C 180,E1 -2863.948,E2 -2863.948} C_VEL
LIN {X 0,Y 559.176,Z 514.828,A -85,B 0,C 180,E1 -2866.185,E2 -2866.185} C_VEL
LIN {X 0,Y 559.2,Z 514.824,A -85,B 0,C 180,E1 -2869.134,E2 -2869.134} C_VEL
LIN {X 0,Y 559.209,Z 514.826,A -85,B 0,C 180,E1 -2872.054,E2 -2872.054} C_VEL
LIN {X 0,Y 559.258,Z 514.815,A -85,B 0,C 180,E1 -2874.954,E2 -2874.954} C_VEL
LIN {X 0,Y 559.257,Z 514.825,A -85,B 0,C 180,E1 -2877.84,E2 -2877.84} C_VEL
LIN {X 0,Y 559.278,Z 514.813,A -85,B 0,C 180,E1 -2880.72,E2 -2880.72} C_VEL
LIN {X 0,Y 559.244,Z 514.817,A -85,B 0,C 180,E1 -2882.882,E2 -2882.882} C_VEL
LIN {X 0,Y 559.234,Z 514.827,A -85,B 0,C 180,E1 -2885.77,E2 -2885.77} C_VEL
LIN {X 0,Y 559.192,Z 514.824,A -85,B 0,C 180,E1 -2888.675,E2 -2888.675} C_VEL
LIN {X 0,Y 559.213,Z 514.826,A -85,B 0,C 180,E1 -2891.601,E2 -2891.601} C_VEL
LIN {X 0,Y 559.208,Z 514.823,A -85,B 0,C 180,E1 -2894.596,E2 -2894.596} C_VEL
LIN {X 0,Y 559.149,Z 514.832,A -85,B 0,C 180,E1 -2897.558,E2 -2897.558} C_VEL
LIN {X 0,Y 559.173,Z 514.833,A -85,B 0,C 180,E1 -2899.838,E2 -2899.838} C_VEL
LIN {X 0,Y 559.149,Z 514.838,A -85,B 0,C 180,E1 -2902.153,E2 -2902.153} C_VEL
LIN {X 0,Y 559.184,Z 514.825,A -85,B 0,C 180,E1 -2905.298,E2 -2905.298} C_VEL
LIN {X 0,Y 559.176,Z 514.831,A -85,B 0,C 180,E1 -2908.381,E2 -2908.381} C_VEL
LIN {X 0,Y 559.153,Z 514.828,A -85,B 0,C 180,E1 -2911.273,E2 -2911.273} C_VEL
LIN {X 0,Y 559.164,Z 514.833,A -85,B 0,C 180,E1 -2913.948,E2 -2913.948} C_VEL
LIN {X 0,Y 559.165,Z 514.833,A -85,B 0,C 180,E1 -2916.447,E2 -2916.447} C_VEL
LIN {X 0,Y 559.181,Z 514.826,A -85,B 0,C 180,E1 -2918.934,E2 -2918.934} C_VEL
LIN {X 0,Y 559.169,Z 514.829,A -85,B 0,C 180,E1 -2921.77,E2 -2921.77} C_VEL
LIN {X 0,Y 559.136,Z 514.834,A -85,B 0,C 180,E1 -2924.74,E2 -2924.74} C_VEL
LIN {X 0,Y 559.167,Z 514.827,A -85,B 0,C 180,E1 -2927.256,E2 -2927.256} C_VEL
LIN {X 0,Y 559.186,Z 514.831,A -85,B 0,C 180,E1 -2930.134,E2 -2930.134} C_VEL
LIN {X 0,Y 559.147,Z 514.831,A -85,B 0,C 180,E1 -2932.891,E2 -2932.891} C_VEL
LIN {X 0,Y 559.173,Z 514.83,A -85,B 0,C 180,E1 -2936.05,E2 -2936.05} C_VEL
LIN {X 0,Y 559.162,Z 514.83,A -85,B 0,C 180,E1 -2938.98,E2 -2938.98} C_VEL
LIN {X 0,Y 559.175,Z 514.827,A -85,B 0,C 180,E1 -2941.618,E2 -2941.618} C_VEL
LIN {X 0,Y 559.184,Z 514.828,A -85,B 0,C 180,E1 -2943.902,E2 -2943.902} C_VEL
LIN {X 0,Y 559.165,Z 514.956,A -85,B 0,C 180,E1 -2946.612,E2 -2946.612} C_VEL
LIN {X 0,Y 560.141,Z 520.502,A -85,B 0,C 180,E1 -2947.499,E2 -2947.499} C_VEL
LIN {X 0,Y 559.83,Z 539.763,A -85,B 0,C 180,E1 -2950.429,E2 -2950.429} C_VEL
LIN {X 0,Y 559.589,Z 556.387,A -85,B 0,C 180,E1 -2952.922,E2 -2952.922} C_VEL
LIN {X 0,Y 559.39,Z 576.069,A -85,B 0,C 180,E1 -2955.818,E2 -2955.818} C_VEL
LIN {X 0,Y 560.313,Z 583.224,A -85,B 0,C 180,E1 -2955.934,E2 -2955.934} C_VEL
LIN {X 0,Y 560.02,Z 683.899,A -85,B 0,C 180,E1 -2957.243,E2 -2957.243} C_VEL
LIN {X 0,Y 559.921,Z 697.187,A -85,B 0,C 180,E1 -2957.563,E2 -2957.563} C_VEL
LIN {X 0,Y 559.81,Z 709.353,A -85,B 0,C 180,E1 -2957.998,E2 -2957.998} C_VEL
LIN {X 0,Y 559.631,Z 721.177,A -85,B 0,C 180,E1 -2958.566,E2 -2958.566} C_VEL
LIN {X 0,Y 559.486,Z 733.186,A -85,B 0,C 180,E1 -2959.321,E2 -2959.321} C_VEL
LIN {X 0,Y 559.299,Z 743.591,A -85,B 0,C 180,E1 -2960.141,E2 -2960.141} C_VEL
LIN {X 0,Y 559.162,Z 752.103,A -85,B 0,C 180,E1 -2960.96,E2 -2960.96} C_VEL
LIN {X 0,Y 559.05,Z 759.953,A -85,B 0,C 180,E1 -2961.869,E2 -2961.869} C_VEL
LIN {X 0,Y 558.936,Z 767.727,A -85,B 0,C 180,E1 -2962.975,E2 -2962.975} C_VEL
LIN {X 0,Y 558.936,Z 774.675,A -85,B 0,C 180,E1 -2964.226,E2 -2964.226} C_VEL
LIN {X 0,Y 558.827,Z 779.368,A -85,B 0,C 180,E1 -2965.31,E2 -2965.31} C_VEL
LIN {X 0,Y 558.836,Z 782.955,A -85,B 0,C 180,E1 -2966.394,E2 -2966.394} C_VEL
LIN {X 0,Y 558.799,Z 784.806,A -85,B 0,C 180,E1 -2967.115,E2 -2967.115} C_VEL
LIN {X 0,Y 558.745,Z 787.184,A -85,B 0,C 180,E1 -2968.557,E2 -2968.557} C_VEL
LIN {X 0,Y 558.74,Z 788,A -85,B 0,C 180,E1 -2969.999,E2 -2969.999} C_VEL
LIN {X 0,Y 558.745,Z 787.187,A -85,B 0,C 180,E1 -2971.44,E2 -2971.44} C_VEL
LIN {X 0,Y 558.799,Z 784.812,A -85,B 0,C 180,E1 -2972.883,E2 -2972.883} C_VEL
LIN {X 0,Y 558.843,Z 781.899,A -85,B 0,C 180,E1 -2973.965,E2 -2973.965} C_VEL
LIN {X 0,Y 558.798,Z 777.953,A -85,B 0,C 180,E1 -2975.05,E2 -2975.05} C_VEL
LIN {X 0,Y 558.917,Z 772.872,A -85,B 0,C 180,E1 -2976.134,E2 -2976.134} C_VEL
LIN {X 0,Y 558.977,Z 766.475,A -85,B 0,C 180,E1 -2977.222,E2 -2977.222} C_VEL
LIN {X 0,Y 559.098,Z 758.487,A -85,B 0,C 180,E1 -2978.311,E2 -2978.311} C_VEL
LIN {X 0,Y 559.184,Z 750.346,A -85,B 0,C 180,E1 -2979.22,E2 -2979.22} C_VEL
LIN {X 0,Y 559.352,Z 740.414,A -85,B 0,C 180,E1 -2980.13,E2 -2980.13} C_VEL
LIN {X 0,Y 559.535,Z 729.381,A -85,B 0,C 180,E1 -2980.938,E2 -2980.938} C_VEL
LIN {X 0,Y 559.702,Z 717.164,A -85,B 0,C 180,E1 -2981.643,E2 -2981.643} C_VEL
LIN {X 0,Y 559.819,Z 704.8,A -85,B 0,C 180,E1 -2982.183,E2 -2982.183} C_VEL
LIN {X 0,Y 559.98,Z 691.393,A -85,B 0,C 180,E1 -2982.594,E2 -2982.594} C_VEL
LIN {X 0,Y 560.101,Z 678.165,A -85,B 0,C 180,E1 -2982.845,E2 -2982.845} C_VEL
LIN {X 0,Y 560.2,Z 581.374,A -85,B 0,C 180,E1 -2984.093,E2 -2984.093} C_VEL
LIN {X 0,Y 559.389,Z 575.8,A -85,B 0,C 180,E1 -2984.203,E2 -2984.203} C_VEL
LIN {X 0,Y 559.622,Z 554.495,A -85,B 0,C 180,E1 -2987.36,E2 -2987.36} C_VEL
LIN {X 0,Y 559.939,Z 534.4,A -85,B 0,C 180,E1 -2990.382,E2 -2990.382} C_VEL
LIN {X 0,Y 560.176,Z 520.516,A -85,B 0,C 180,E1 -2992.497,E2 -2992.497} C_VEL
LIN {X 0,Y 559.171,Z 514.839,A -85,B 0,C 180,E1 -2993.435,E2 -2993.435} C_VEL
LIN {X 0,Y 559.179,Z 514.829,A -85,B 0,C 180,E1 -2996.096,E2 -2996.096} C_VEL
LIN {X 0,Y 559.161,Z 514.83,A -85,B 0,C 180,E1 -2998.528,E2 -2998.528} C_VEL
LIN {X 0,Y 559.152,Z 514.837,A -85,B 0,C 180,E1 -3001.273,E2 -3001.273} C_VEL
LIN {X 0,Y 559.163,Z 514.831,A -85,B 0,C 180,E1 -3003.948,E2 -3003.948} C_VEL
LIN {X 0,Y 559.141,Z 514.835,A -85,B 0,C 180,E1 -3007.107,E2 -3007.107} C_VEL
LIN {X 0,Y 559.165,Z 514.831,A -85,B 0,C 180,E1 -3009.942,E2 -3009.942} C_VEL
LIN {X 0,Y 559.159,Z 514.83,A -85,B 0,C 180,E1 -3012.742,E2 -3012.742} C_VEL
LIN {X 0,Y 559.146,Z 514.836,A -85,B 0,C 180,E1 -3015.76,E2 -3015.76} C_VEL
LIN {X 0,Y 559.185,Z 514.826,A -85,B 0,C 180,E1 -3018.231,E2 -3018.231} C_VEL
LIN {X 0,Y 559.171,Z 514.832,A -85,B 0,C 180,E1 -3021.19,E2 -3021.19} C_VEL
LIN {X 0,Y 559.166,Z 514.832,A -85,B 0,C 180,E1 -3023.791,E2 -3023.791} C_VEL
LIN {X 0,Y 559.17,Z 514.826,A -85,B 0,C 180,E1 -3026.425,E2 -3026.425} C_VEL
LIN {X 0,Y 559.158,Z 514.831,A -85,B 0,C 180,E1 -3028.981,E2 -3028.981} C_VEL
LIN {X 0,Y 559.163,Z 514.834,A -85,B 0,C 180,E1 -3031.617,E2 -3031.617} C_VEL
LIN {X 0,Y 559.191,Z 514.827,A -85,B 0,C 180,E1 -3033.903,E2 -3033.903} C_VEL
LIN {X 0,Y 559.147,Z 514.828,A -85,B 0,C 180,E1 -3036.566,E2 -3036.566} C_VEL
LIN {X 0,Y 559.177,Z 514.836,A -85,B 0,C 180,E1 -3039.395,E2 -3039.395} C_VEL
LIN {X 0,Y 559.147,Z 514.836,A -85,B 0,C 180,E1 -3041.685,E2 -3041.685} C_VEL
LIN {X 0,Y 559.161,Z 514.829,A -85,B 0,C 180,E1 -3043.947,E2 -3043.947} C_VEL
LIN {X 0,Y 559.164,Z 514.828,A -85,B 0,C 180,E1 -3046.184,E2 -3046.184} C_VEL
LIN {X 0,Y 559.201,Z 514.827,A -85,B 0,C 180,E1 -3049.133,E2 -3049.133} C_VEL
LIN {X 0,Y 559.2,Z 514.824,A -85,B 0,C 180,E1 -3052.053,E2 -3052.053} C_VEL
LIN {X 0,Y 559.252,Z 514.819,A -85,B 0,C 180,E1 -3054.953,E2 -3054.953} C_VEL
LIN {X 0,Y 559.242,Z 514.821,A -85,B 0,C 180,E1 -3057.839,E2 -3057.839} C_VEL
LIN {X 0,Y 559.267,Z 514.816,A -85,B 0,C 180,E1 -3060.72,E2 -3060.72} C_VEL
LIN {X 0,Y 559.236,Z 514.821,A -85,B 0,C 180,E1 -3062.881,E2 -3062.881} C_VEL
LIN {X 0,Y 559.22,Z 514.825,A -85,B 0,C 180,E1 -3065.77,E2 -3065.77} C_VEL
LIN {X 0,Y 559.193,Z 514.825,A -85,B 0,C 180,E1 -3068.674,E2 -3068.674} C_VEL
LIN {X 0,Y 559.197,Z 514.831,A -85,B 0,C 180,E1 -3071.6,E2 -3071.6} C_VEL
LIN {X 0,Y 559.187,Z 514.826,A -85,B 0,C 180,E1 -3074.595,E2 -3074.595} C_VEL
LIN {X 0,Y 559.153,Z 514.837,A -85,B 0,C 180,E1 -3077.557,E2 -3077.557} C_VEL
LIN {X 0,Y 559.164,Z 514.831,A -85,B 0,C 180,E1 -3079.837,E2 -3079.837} C_VEL
LIN {X 0,Y 559.132,Z 514.833,A -85,B 0,C 180,E1 -3082.153,E2 -3082.153} C_VEL
LIN {X 0,Y 559.167,Z 514.835,A -85,B 0,C 180,E1 -3085.188,E2 -3085.188} C_VEL
LIN {X 0,Y 559.184,Z 514.833,A -85,B 0,C 180,E1 -3087.712,E2 -3087.712} C_VEL
LIN {X 0,Y 559.155,Z 514.837,A -85,B 0,C 180,E1 -3089.54,E2 -3089.54} C_VEL
LIN {X 0,Y 558.861,Z 515.383,A -85,B 0,C 180,E1 -3089.937,E2 -3089.937} C_VEL
LIN {X 0,Y 557.606,Z 517.638,A -85,B 0,C 180,E1 -3090.492,E2 -3090.492} C_VEL
LIN {X 0,Y 553.566,Z 524.82,A -85,B 0,C 180,E1 -3091.678,E2 -3091.678} C_VEL
LIN {X 0,Y 552.548,Z 527.867,A -85,B 0,C 180,E1 -3092.202,E2 -3092.202} C_VEL
LIN {X 0,Y 552.457,Z 528.865,A -85,B 0,C 180,E1 -3092.381,E2 -3092.381} C_VEL
LIN {X 0,Y 552.234,Z 544.466,A -85,B 0,C 180,E1 -3095.199,E2 -3095.199} C_VEL
LIN {X 0,Y 552.199,Z 547.097,A -85,B 0,C 180,E1 -3095.671,E2 -3095.671} C_VEL
LIN {X 0,Y 553.431,Z 555.208,A -85,B 0,C 180,E1 -3095.827,E2 -3095.827} C_VEL
LIN {X 0,Y 553.113,Z 654.696,A -85,B 0,C 180,E1 -3097.142,E2 -3097.142} C_VEL
LIN {X 0,Y 552.937,Z 668.582,A -85,B 0,C 180,E1 -3097.492,E2 -3097.492} C_VEL
LIN {X 0,Y 552.786,Z 681.447,A -85,B 0,C 180,E1 -3097.98,E2 -3097.98} C_VEL
LIN {X 0,Y 552.609,Z 693.787,A -85,B 0,C 180,E1 -3098.616,E2 -3098.616} C_VEL
LIN {X 0,Y 552.412,Z 705.398,A -85,B 0,C 180,E1 -3099.389,E2 -3099.389} C_VEL
LIN {X 0,Y 552.23,Z 716.42,A -85,B 0,C 180,E1 -3100.318,E2 -3100.318} C_VEL
LIN {X 0,Y 552.086,Z 725.951,A -85,B 0,C 180,E1 -3101.32,E2 -3101.32} C_VEL
LIN {X 0,Y 551.9,Z 734.592,A -85,B 0,C 180,E1 -3102.447,E2 -3102.447} C_VEL
LIN {X 0,Y 551.825,Z 742.179,A -85,B 0,C 180,E1 -3103.702,E2 -3103.702} C_VEL
LIN {X 0,Y 551.777,Z 748.311,A -85,B 0,C 180,E1 -3105.019,E2 -3105.019} C_VEL
LIN {X 0,Y 551.726,Z 751.92,A -85,B 0,C 180,E1 -3106.036,E2 -3106.036} C_VEL
LIN {X 0,Y 551.674,Z 754.622,A -85,B 0,C 180,E1 -3107.047,E2 -3107.047} C_VEL
LIN {X 0,Y 551.652,Z 755.828,A -85,B 0,C 180,E1 -3107.638,E2 -3107.638} C_VEL
LIN {X 0,Y 551.657,Z 757.342,A -85,B 0,C 180,E1 -3108.733,E2 -3108.733} C_VEL
LIN {X 0,Y 551.637,Z 757.966,A -85,B 0,C 180,E1 -3109.854,E2 -3109.854} C_VEL
LIN {X 0,Y 551.633,Z 757.64,A -85,B 0,C 180,E1 -3111.001,E2 -3111.001} C_VEL
LIN {X 0,Y 551.649,Z 756.101,A -85,B 0,C 180,E1 -3112.302,E2 -3112.302} C_VEL
LIN {X 0,Y 551.756,Z 752.786,A -85,B 0,C 180,E1 -3113.758,E2 -3113.758} C_VEL
LIN {X 0,Y 551.712,Z 748.491,A -85,B 0,C 180,E1 -3115.026,E2 -3115.026} C_VEL
LIN {X 0,Y 551.829,Z 742.33,A -85,B 0,C 180,E1 -3116.359,E2 -3116.359} C_VEL
LIN {X 0,Y 551.899,Z 736.005,A -85,B 0,C 180,E1 -3117.432,E2 -3117.432} C_VEL
LIN {X 0,Y 552.034,Z 727.911,A -85,B 0,C 180,E1 -3118.537,E2 -3118.537} C_VEL
LIN {X 0,Y 552.174,Z 718.765,A -85,B 0,C 180,E1 -3119.544,E2 -3119.544} C_VEL
LIN {X 0,Y 552.334,Z 708.522,A -85,B 0,C 180,E1 -3120.459,E2 -3120.459} C_VEL
LIN {X 0,Y 552.531,Z 697.293,A -85,B 0,C 180,E1 -3121.259,E2 -3121.259} C_VEL
LIN {X 0,Y 552.764,Z 685.122,A -85,B 0,C 180,E1 -3121.939,E2 -3121.939} C_VEL
LIN {X 0,Y 552.909,Z 672.619,A -85,B 0,C 180,E1 -3122.462,E2 -3122.462} C_VEL
LIN {X 0,Y 553.091,Z 659.779,A -85,B 0,C 180,E1 -3122.841,E2 -3122.841} C_VEL
LIN {X 0,Y 553.171,Z 646.371,A -85,B 0,C 180,E1 -3123.077,E2 -3123.077} C_VEL
LIN {X 0,Y 553.286,Z 553.588,A -85,B 0,C 180,E1 -3124.288,E2 -3124.288} C_VEL
LIN {X 0,Y 552.198,Z 547.173,A -85,B 0,C 180,E1 -3124.405,E2 -3124.405} C_VEL
LIN {X 0,Y 552.459,Z 530.731,A -85,B 0,C 180,E1 -3127.369,E2 -3127.369} C_VEL
LIN {X 0,Y 552.568,Z 518.929,A -85,B 0,C 180,E1 -3129.528,E2 -3129.528} C_VEL
LIN {X 0,Y 552.154,Z 515.709,A -85,B 0,C 180,E1 -3130.184,E2 -3130.184} C_VEL
LIN {X 0,Y 552.151,Z 515.709,A -85,B 0,C 180,E1 -3132.978,E2 -3132.978} C_VEL
LIN {X 0,Y 552.133,Z 515.704,A -85,B 0,C 180,E1 -3136.006,E2 -3136.006} C_VEL
LIN {X 0,Y 552.158,Z 515.707,A -85,B 0,C 180,E1 -3138.994,E2 -3138.994} C_VEL
LIN {X 0,Y 552.156,Z 515.7,A -85,B 0,C 180,E1 -3141.953,E2 -3141.953} C_VEL
LIN {X 0,Y 552.228,Z 515.701,A -85,B 0,C 180,E1 -3144.89,E2 -3144.89} C_VEL
LIN {X 0,Y 552.224,Z 515.691,A -85,B 0,C 180,E1 -3147.813,E2 -3147.813} C_VEL
LIN {X 0,Y 552.242,Z 515.696,A -85,B 0,C 180,E1 -3150.73,E2 -3150.73} C_VEL
LIN {X 0,Y 552.203,Z 515.704,A -85,B 0,C 180,E1 -3152.919,E2 -3152.919} C_VEL
LIN {X 0,Y 552.198,Z 515.695,A -85,B 0,C 180,E1 -3155.845,E2 -3155.845} C_VEL
LIN {X 0,Y 552.156,Z 515.706,A -85,B 0,C 180,E1 -3158.787,E2 -3158.787} C_VEL
LIN {X 0,Y 552.162,Z 515.7,A -85,B 0,C 180,E1 -3161.751,E2 -3161.751} C_VEL
LIN {X 0,Y 552.136,Z 515.707,A -85,B 0,C 180,E1 -3164.749,E2 -3164.749} C_VEL
LIN {X 0,Y 552.1,Z 515.708,A -85,B 0,C 180,E1 -3167.79,E2 -3167.79} C_VEL
LIN {X 0,Y 552.131,Z 515.703,A -85,B 0,C 180,E1 -3170.102,E2 -3170.102} C_VEL
LIN {X 0,Y 552.092,Z 515.709,A -85,B 0,C 180,E1 -3172.452,E2 -3172.452} C_VEL
LIN {X 0,Y 552.156,Z 515.707,A -85,B 0,C 180,E1 -3175.351,E2 -3175.351} C_VEL
LIN {X 0,Y 552.11,Z 515.706,A -85,B 0,C 180,E1 -3178.099,E2 -3178.099} C_VEL
LIN {X 0,Y 552.109,Z 515.707,A -85,B 0,C 180,E1 -3180.61,E2 -3180.61} C_VEL
LIN {X 0,Y 552.117,Z 515.714,A -85,B 0,C 180,E1 -3183.187,E2 -3183.187} C_VEL
LIN {X 0,Y 552.087,Z 515.711,A -85,B 0,C 180,E1 -3185.845,E2 -3185.845} C_VEL
LIN {X 0,Y 552.127,Z 515.709,A -85,B 0,C 180,E1 -3189.063,E2 -3189.063} C_VEL
LIN {X 0,Y 552.142,Z 515.71,A -85,B 0,C 180,E1 -3191.445,E2 -3191.445} C_VEL
LIN {X 0,Y 552.099,Z 515.707,A -85,B 0,C 180,E1 -3194.533,E2 -3194.533} C_VEL
LIN {X 0,Y 552.132,Z 515.71,A -85,B 0,C 180,E1 -3197.585,E2 -3197.585} C_VEL
LIN {X 0,Y 552.135,Z 515.703,A -85,B 0,C 180,E1 -3200.474,E2 -3200.474} C_VEL
LIN {X 0,Y 552.109,Z 515.714,A -85,B 0,C 180,E1 -3203.318,E2 -3203.318} C_VEL
LIN {X 0,Y 552.133,Z 515.706,A -85,B 0,C 180,E1 -3205.94,E2 -3205.94} C_VEL
LIN {X 0,Y 552.123,Z 515.704,A -85,B 0,C 180,E1 -3208.541,E2 -3208.541} C_VEL
LIN {X 0,Y 552.129,Z 515.712,A -85,B 0,C 180,E1 -3211.439,E2 -3211.439} C_VEL
LIN {X 0,Y 552.135,Z 515.703,A -85,B 0,C 180,E1 -3214.356,E2 -3214.356} C_VEL
LIN {X 0,Y 552.101,Z 515.707,A -85,B 0,C 180,E1 -3216.758,E2 -3216.758} C_VEL
LIN {X 0,Y 552.123,Z 515.707,A -85,B 0,C 180,E1 -3219.12,E2 -3219.12} C_VEL
LIN {X 0,Y 552.126,Z 515.711,A -85,B 0,C 180,E1 -3221.445,E2 -3221.445} C_VEL
LIN {X 0,Y 552.122,Z 515.713,A -85,B 0,C 180,E1 -3223.738,E2 -3223.738} C_VEL
LIN {X 0,Y 552.14,Z 515.707,A -85,B 0,C 180,E1 -3226.005,E2 -3226.005} C_VEL
LIN {X 0,Y 552.168,Z 515.699,A -85,B 0,C 180,E1 -3228.994,E2 -3228.994} C_VEL
LIN {X 0,Y 552.163,Z 515.706,A -85,B 0,C 180,E1 -3231.952,E2 -3231.952} C_VEL
LIN {X 0,Y 552.233,Z 515.69,A -85,B 0,C 180,E1 -3234.889,E2 -3234.889} C_VEL
LIN {X 0,Y 552.228,Z 515.701,A -85,B 0,C 180,E1 -3237.812,E2 -3237.812} C_VEL
LIN {X 0,Y 552.248,Z 515.689,A -85,B 0,C 180,E1 -3240.73,E2 -3240.73} C_VEL
LIN {X 0,Y 552.211,Z 515.693,A -85,B 0,C 180,E1 -3242.918,E2 -3242.918} C_VEL
LIN {X 0,Y 552.205,Z 515.704,A -85,B 0,C 180,E1 -3245.844,E2 -3245.844} C_VEL
LIN {X 0,Y 552.159,Z 515.7,A -85,B 0,C 180,E1 -3248.786,E2 -3248.786} C_VEL
LIN {X 0,Y 552.17,Z 515.705,A -85,B 0,C 180,E1 -3251.751,E2 -3251.751} C_VEL
LIN {X 0,Y 552.144,Z 515.702,A -85,B 0,C 180,E1 -3254.749,E2 -3254.749} C_VEL
LIN {X 0,Y 552.107,Z 515.713,A -85,B 0,C 180,E1 -3257.789,E2 -3257.789} C_VEL
LIN {X 0,Y 552.134,Z 515.712,A -85,B 0,C 180,E1 -3260.101,E2 -3260.101} C_VEL
LIN {X 0,Y 552.099,Z 515.711,A -85,B 0,C 180,E1 -3262.451,E2 -3262.451} C_VEL
LIN {X 0,Y 552.163,Z 515.7,A -85,B 0,C 180,E1 -3265.35,E2 -3265.35} C_VEL
LIN {X 0,Y 552.114,Z 515.716,A -85,B 0,C 180,E1 -3268.098,E2 -3268.098} C_VEL
LIN {X 0,Y 552.109,Z 515.709,A -85,B 0,C 180,E1 -3270.609,E2 -3270.609} C_VEL
LIN {X 0,Y 552.114,Z 515.705,A -85,B 0,C 180,E1 -3273.186,E2 -3273.186} C_VEL
LIN {X 0,Y 552.108,Z 515.71,A -85,B 0,C 180,E1 -3275.842,E2 -3275.842} C_VEL
LIN {X 0,Y 552.129,Z 515.704,A -85,B 0,C 180,E1 -3279.061,E2 -3279.061} C_VEL
LIN {X 0,Y 552.127,Z 515.704,A -85,B 0,C 180,E1 -3281.446,E2 -3281.446} C_VEL
LIN {X 0,Y 552.085,Z 515.715,A -85,B 0,C 180,E1 -3284.53,E2 -3284.53} C_VEL
LIN {X 0,Y 552.137,Z 515.703,A -85,B 0,C 180,E1 -3287.584,E2 -3287.584} C_VEL
LIN {X 0,Y 552.136,Z 515.71,A -85,B 0,C 180,E1 -3290.472,E2 -3290.472} C_VEL
LIN {X 0,Y 552.113,Z 515.705,A -85,B 0,C 180,E1 -3293.317,E2 -3293.317} C_VEL
LIN {X 0,Y 552.133,Z 515.706,A -85,B 0,C 180,E1 -3295.939,E2 -3295.939} C_VEL
LIN {X 0,Y 552.126,Z 515.713,A -85,B 0,C 180,E1 -3298.54,E2 -3298.54} C_VEL
LIN {X 0,Y 552.131,Z 515.704,A -85,B 0,C 180,E1 -3301.437,E2 -3301.437} C_VEL
LIN {X 0,Y 552.135,Z 515.712,A -85,B 0,C 180,E1 -3304.355,E2 -3304.355} C_VEL
LIN {X 0,Y 552.138,Z 515.896,A -85,B 0,C 180,E1 -3306.467,E2 -3306.467} C_VEL
LIN {X 0,Y 553.177,Z 521.611,A -85,B 0,C 180,E1 -3307.398,E2 -3307.398} C_VEL
LIN {X 0,Y 552.915,Z 539.631,A -85,B 0,C 180,E1 -3310.153,E2 -3310.153} C_VEL
LIN {X 0,Y 552.622,Z 557.129,A -85,B 0,C 180,E1 -3312.812,E2 -3312.812} C_VEL
LIN {X 0,Y 552.361,Z 575.892,A -85,B 0,C 180,E1 -3315.626,E2 -3315.626} C_VEL
LIN {X 0,Y 553.45,Z 583.769,A -85,B 0,C 180,E1 -3315.763,E2 -3315.763} C_VEL
LIN {X 0,Y 553.108,Z 683.899,A -85,B 0,C 180,E1 -3317.081,E2 -3317.081} C_VEL
LIN {X 0,Y 553.001,Z 697.186,A -85,B 0,C 180,E1 -3317.405,E2 -3317.405} C_VEL
LIN {X 0,Y 552.853,Z 709.346,A -85,B 0,C 180,E1 -3317.845,E2 -3317.845} C_VEL
LIN {X 0,Y 552.662,Z 720.16,A -85,B 0,C 180,E1 -3318.365,E2 -3318.365} C_VEL
LIN {X 0,Y 552.533,Z 731.893,A -85,B 0,C 180,E1 -3319.093,E2 -3319.093} C_VEL
LIN {X 0,Y 552.292,Z 742.528,A -85,B 0,C 180,E1 -3319.922,E2 -3319.922} C_VEL
LIN {X 0,Y 552.126,Z 752.103,A -85,B 0,C 180,E1 -3320.844,E2 -3320.844} C_VEL
LIN {X 0,Y 552.013,Z 759.953,A -85,B 0,C 180,E1 -3321.764,E2 -3321.764} C_VEL
LIN {X 0,Y 551.889,Z 767.615,A -85,B 0,C 180,E1 -3322.867,E2 -3322.867} C_VEL
LIN {X 0,Y 551.867,Z 774.675,A -85,B 0,C 180,E1 -3324.152,E2 -3324.152} C_VEL
LIN {X 0,Y 551.725,Z 779.369,A -85,B 0,C 180,E1 -3325.25,E2 -3325.25} C_VEL
LIN {X 0,Y 551.751,Z 782.955,A -85,B 0,C 180,E1 -3326.347,E2 -3326.347} C_VEL
LIN {X 0,Y 551.724,Z 784.805,A -85,B 0,C 180,E1 -3327.078,E2 -3327.078} C_VEL
LIN {X 0,Y 551.645,Z 787.183,A -85,B 0,C 180,E1 -3328.539,E2 -3328.539} C_VEL
LIN {X 0,Y 551.64,Z 788,A -85,B 0,C 180,E1 -3329.999,E2 -3329.999} C_VEL
LIN {X 0,Y 551.645,Z 787.186,A -85,B 0,C 180,E1 -3331.459,E2 -3331.459} C_VEL
LIN {X 0,Y 551.723,Z 784.812,A -85,B 0,C 180,E1 -3332.92,E2 -3332.92} C_VEL
LIN {X 0,Y 551.763,Z 781.899,A -85,B 0,C 180,E1 -3334.016,E2 -3334.016} C_VEL
LIN {X 0,Y 551.724,Z 777.953,A -85,B 0,C 180,E1 -3335.115,E2 -3335.115} C_VEL
LIN {X 0,Y 551.813,Z 772.136,A -85,B 0,C 180,E1 -3336.351,E2 -3336.351} C_VEL
LIN {X 0,Y 551.926,Z 765.244,A -85,B 0,C 180,E1 -3337.498,E2 -3337.498} C_VEL
LIN {X 0,Y 552.081,Z 757,A -85,B 0,C 180,E1 -3338.601,E2 -3338.601} C_VEL
LIN {X 0,Y 552.221,Z 748.551,A -85,B 0,C 180,E1 -3339.522,E2 -3339.522} C_VEL
LIN {X 0,Y 552.411,Z 738.11,A -85,B 0,C 180,E1 -3340.444,E2 -3340.444} C_VEL
LIN {X 0,Y 552.589,Z 727.148,A -85,B 0,C 180,E1 -3341.223,E2 -3341.223} C_VEL
LIN {X 0,Y 552.782,Z 716.429,A -85,B 0,C 180,E1 -3341.829,E2 -3341.829} C_VEL
LIN {X 0,Y 552.901,Z 704.796,A -85,B 0,C 180,E1 -3342.338,E2 -3342.338} C_VEL
LIN {X 0,Y 553.057,Z 691.392,A -85,B 0,C 180,E1 -3342.754,E2 -3342.754} C_VEL
LIN {X 0,Y 553.188,Z 678.165,A -85,B 0,C 180,E1 -3343.008,E2 -3343.008} C_VEL
LIN {X 0,Y 553.319,Z 582.087,A -85,B 0,C 180,E1 -3344.262,E2 -3344.262} C_VEL
LIN {X 0,Y 552.377,Z 575.772,A -85,B 0,C 180,E1 -3344.392,E2 -3344.392} C_VEL
LIN {X 0,Y 552.663,Z 555.103,A -85,B 0,C 180,E1 -3347.494,E2 -3347.494} C_VEL
LIN {X 0,Y 553.019,Z 534.367,A -85,B 0,C 180,E1 -3350.649,E2 -3350.649} C_VEL
LIN {X 0,Y 553.212,Z 521.619,A -85,B 0,C 180,E1 -3352.599,E2 -3352.599} C_VEL
LIN {X 0,Y 552.121,Z 515.716,A -85,B 0,C 180,E1 -3353.58,E2 -3353.58} C_VEL
LIN {X 0,Y 552.118,Z 515.707,A -85,B 0,C 180,E1 -3356.455,E2 -3356.455} C_VEL
LIN {X 0,Y 552.108,Z 515.711,A -85,B 0,C 180,E1 -3358.927,E2 -3358.927} C_VEL
LIN {X 0,Y 552.133,Z 515.714,A -85,B 0,C 180,E1 -3361.479,E2 -3361.479} C_VEL
LIN {X 0,Y 552.131,Z 515.705,A -85,B 0,C 180,E1 -3364.169,E2 -3364.169} C_VEL
LIN {X 0,Y 552.106,Z 515.708,A -85,B 0,C 180,E1 -3366.745,E2 -3366.745} C_VEL
LIN {X 0,Y 552.146,Z 515.712,A -85,B 0,C 180,E1 -3369.524,E2 -3369.524} C_VEL
LIN {X 0,Y 552.125,Z 515.705,A -85,B 0,C 180,E1 -3372.424,E2 -3372.424} C_VEL
LIN {X 0,Y 552.092,Z 515.718,A -85,B 0,C 180,E1 -3375.562,E2 -3375.562} C_VEL
LIN {X 0,Y 552.133,Z 515.704,A -85,B 0,C 180,E1 -3378.675,E2 -3378.675} C_VEL
LIN {X 0,Y 552.113,Z 515.715,A -85,B 0,C 180,E1 -3381.41,E2 -3381.41} C_VEL
LIN {X 0,Y 552.107,Z 515.708,A -85,B 0,C 180,E1 -3384.158,E2 -3384.158} C_VEL
LIN {X 0,Y 552.121,Z 515.706,A -85,B 0,C 180,E1 -3386.814,E2 -3386.814} C_VEL
LIN {X 0,Y 552.106,Z 515.715,A -85,B 0,C 180,E1 -3389.391,E2 -3389.391} C_VEL
LIN {X 0,Y 552.119,Z 515.707,A -85,B 0,C 180,E1 -3391.902,E2 -3391.902} C_VEL
LIN {X 0,Y 552.148,Z 515.702,A -85,B 0,C 180,E1 -3394.648,E2 -3394.648} C_VEL
LIN {X 0,Y 552.087,Z 515.717,A -85,B 0,C 180,E1 -3397.548,E2 -3397.548} C_VEL
LIN {X 0,Y 552.139,Z 515.701,A -85,B 0,C 180,E1 -3400.372,E2 -3400.372} C_VEL
LIN {X 0,Y 552.148,Z 515.705,A -85,B 0,C 180,E1 -3402.977,E2 -3402.977} C_VEL
LIN {X 0,Y 552.126,Z 515.706,A -85,B 0,C 180,E1 -3406.004,E2 -3406.004} C_VEL
LIN {X 0,Y 552.168,Z 515.701,A -85,B 0,C 180,E1 -3408.993,E2 -3408.993} C_VEL
LIN {X 0,Y 552.154,Z 515.702,A -85,B 0,C 180,E1 -3411.951,E2 -3411.951} C_VEL
LIN {X 0,Y 552.225,Z 515.694,A -85,B 0,C 180,E1 -3414.889,E2 -3414.889} C_VEL
LIN {X 0,Y 552.214,Z 515.696,A -85,B 0,C 180,E1 -3417.811,E2 -3417.811} C_VEL
LIN {X 0,Y 552.237,Z 515.692,A -85,B 0,C 180,E1 -3420.729,E2 -3420.729} C_VEL
LIN {X 0,Y 552.202,Z 515.697,A -85,B 0,C 180,E1 -3422.918,E2 -3422.918} C_VEL
LIN {X 0,Y 552.19,Z 515.7,A -85,B 0,C 180,E1 -3425.844,E2 -3425.844} C_VEL
LIN {X 0,Y 552.161,Z 515.702,A -85,B 0,C 180,E1 -3428.785,E2 -3428.785} C_VEL
LIN {X 0,Y 552.153,Z 515.706,A -85,B 0,C 180,E1 -3431.75,E2 -3431.75} C_VEL
LIN {X 0,Y 552.124,Z 515.707,A -85,B 0,C 180,E1 -3434.748,E2 -3434.748} C_VEL
LIN {X 0,Y 552.104,Z 515.712,A -85,B 0,C 180,E1 -3437.788,E2 -3437.788} C_VEL
LIN {X 0,Y 552.123,Z 515.706,A -85,B 0,C 180,E1 -3440.101,E2 -3440.101} C_VEL
LIN {X 0,Y 552.086,Z 515.71,A -85,B 0,C 180,E1 -3442.451,E2 -3442.451} C_VEL
LIN {X 0,Y 552.145,Z 515.711,A -85,B 0,C 180,E1 -3445.351,E2 -3445.351} C_VEL
LIN {X 0,Y 552.116,Z 515.71,A -85,B 0,C 180,E1 -3448.097,E2 -3448.097} C_VEL
LIN {X 0,Y 552.173,Z 515.824,A -85,B 0,C 180,E1 -3449.963,E2 -3449.963} C_VEL
LIN {X 0,Y 552.613,Z 520.147,A -85,B 0,C 180,E1 -3450.789,E2 -3450.789} C_VEL
LIN {X 0,Y 552.457,Z 528.865,A -85,B 0,C 180,E1 -3452.381,E2 -3452.381} C_VEL
LIN {X 0,Y 551.754,Z 531.86,A -85,B 0,C 180,E1 -3452.904,E2 -3452.904} C_VEL
LIN {X 0,Y 545.889,Z 542.027,A -85,B 0,C 180,E1 -3454.578,E2 -3454.578} C_VEL
LIN {X 0,Y 545.205,Z 545.046,A -85,B 0,C 180,E1 -3455.109,E2 -3455.109} C_VEL
LIN {X 0,Y 545.168,Z 547.268,A -85,B 0,C 180,E1 -3455.501,E2 -3455.501} C_VEL
LIN {X 0,Y 546.573,Z 556.283,A -85,B 0,C 180,E1 -3455.659,E2 -3455.659} C_VEL
LIN {X 0,Y 546.223,Z 654.062,A -85,B 0,C 180,E1 -3456.963,E2 -3456.963} C_VEL
LIN {X 0,Y 546.072,Z 666.89,A -85,B 0,C 180,E1 -3457.279,E2 -3457.279} C_VEL
LIN {X 0,Y 545.848,Z 680.069,A -85,B 0,C 180,E1 -3457.762,E2 -3457.762} C_VEL
LIN {X 0,Y 545.666,Z 691.865,A -85,B 0,C 180,E1 -3458.356,E2 -3458.356} C_VEL
LIN {X 0,Y 545.473,Z 702.356,A -85,B 0,C 180,E1 -3459.028,E2 -3459.028} C_VEL
LIN {X 0,Y 545.274,Z 713.489,A -85,B 0,C 180,E1 -3459.919,E2 -3459.919} C_VEL
LIN {X 0,Y 545.075,Z 723.676,A -85,B 0,C 180,E1 -3460.944,E2 -3460.944} C_VEL
LIN {X 0,Y 544.911,Z 731.972,A -85,B 0,C 180,E1 -3461.973,E2 -3461.973} C_VEL
LIN {X 0,Y 544.775,Z 739.509,A -85,B 0,C 180,E1 -3463.136,E2 -3463.136} C_VEL
LIN {X 0,Y 544.723,Z 744.878,A -85,B 0,C 180,E1 -3464.163,E2 -3464.163} C_VEL
LIN {X 0,Y 544.669,Z 749.274,A -85,B 0,C 180,E1 -3465.208,E2 -3465.208} C_VEL
LIN {X 0,Y 544.616,Z 752.758,A -85,B 0,C 180,E1 -3466.273,E2 -3466.273} C_VEL
LIN {X 0,Y 544.569,Z 755.359,A -85,B 0,C 180,E1 -3467.359,E2 -3467.359} C_VEL
LIN {X 0,Y 544.552,Z 757.47,A -85,B 0,C 180,E1 -3468.839,E2 -3468.839} C_VEL
LIN {X 0,Y 544.54,Z 757.958,A -85,B 0,C 180,E1 -3469.812,E2 -3469.812} C_VEL
LIN {X 0,Y 544.542,Z 757.79,A -85,B 0,C 180,E1 -3470.774,E2 -3470.774} C_VEL
LIN {X 0,Y 544.526,Z 756.689,A -85,B 0,C 180,E1 -3471.934,E2 -3471.934} C_VEL
LIN {X 0,Y 544.583,Z 754.479,A -85,B 0,C 180,E1 -3473.141,E2 -3473.141} C_VEL
LIN {X 0,Y 544.626,Z 750.637,A -85,B 0,C 180,E1 -3474.502,E2 -3474.502} C_VEL
LIN {X 0,Y 544.64,Z 746.058,A -85,B 0,C 180,E1 -3475.674,E2 -3475.674} C_VEL
LIN {X 0,Y 544.769,Z 741.093,A -85,B 0,C 180,E1 -3476.675,E2 -3476.675} C_VEL
LIN {X 0,Y 544.86,Z 733.802,A -85,B 0,C 180,E1 -3477.856,E2 -3477.856} C_VEL
LIN {X 0,Y 545.061,Z 725.372,A -85,B 0,C 180,E1 -3478.953,E2 -3478.953} C_VEL
LIN {X 0,Y 545.224,Z 716.097,A -85,B 0,C 180,E1 -3479.929,E2 -3479.929} C_VEL
LIN {X 0,Y 545.407,Z 705.602,A -85,B 0,C 180,E1 -3480.823,E2 -3480.823} C_VEL
LIN {X 0,Y 545.598,Z 695.214,A -85,B 0,C 180,E1 -3481.537,E2 -3481.537} C_VEL
LIN {X 0,Y 545.836,Z 683.315,A -85,B 0,C 180,E1 -3482.178,E2 -3482.178} C_VEL
LIN {X 0,Y 546.026,Z 670.479,A -85,B 0,C 180,E1 -3482.699,E2 -3482.699} C_VEL
LIN {X 0,Y 546.156,Z 657.433,A -85,B 0,C 180,E1 -3483.058,E2 -3483.058} C_VEL
LIN {X 0,Y 546.258,Z 639.074,A -85,B 0,C 180,E1 -3483.342,E2 -3483.342} C_VEL
LIN {X 0,Y 546.403,Z 554.36,A -85,B 0,C 180,E1 -3484.461,E2 -3484.461} C_VEL
LIN {X 0,Y 545.175,Z 547.117,A -85,B 0,C 180,E1 -3484.605,E2 -3484.605} C_VEL
LIN {X 0,Y 545.439,Z 530.422,A -85,B 0,C 180,E1 -3487.661,E2 -3487.661} C_VEL
LIN {X 0,Y 545.572,Z 519.803,A -85,B 0,C 180,E1 -3489.648,E2 -3489.648} C_VEL
LIN {X 0,Y 545.107,Z 516.588,A -85,B 0,C 180,E1 -3490.294,E2 -3490.294} C_VEL
LIN {X 0,Y 545.09,Z 516.591,A -85,B 0,C 180,E1 -3492.751,E2 -3492.751} C_VEL
LIN {X 0,Y 545.092,Z 516.581,A -85,B 0,C 180,E1 -3495.821,E2 -3495.821} C_VEL
LIN {X 0,Y 545.114,Z 516.587,A -85,B 0,C 180,E1 -3498.85,E2 -3498.85} C_VEL
LIN {X 0,Y 545.126,Z 516.576,A -85,B 0,C 180,E1 -3501.848,E2 -3501.848} C_VEL
LIN {X 0,Y 545.203,Z 516.576,A -85,B 0,C 180,E1 -3504.824,E2 -3504.824} C_VEL
LIN {X 0,Y 545.195,Z 516.567,A -85,B 0,C 180,E1 -3507.785,E2 -3507.785} C_VEL
LIN {X 0,Y 545.212,Z 516.572,A -85,B 0,C 180,E1 -3510.74,E2 -3510.74} C_VEL
LIN {X 0,Y 545.17,Z 516.581,A -85,B 0,C 180,E1 -3512.957,E2 -3512.957} C_VEL
LIN {X 0,Y 545.169,Z 516.57,A -85,B 0,C 180,E1 -3515.921,E2 -3515.921} C_VEL
LIN {X 0,Y 545.116,Z 516.585,A -85,B 0,C 180,E1 -3518.901,E2 -3518.901} C_VEL
LIN {X 0,Y 545.134,Z 516.575,A -85,B 0,C 180,E1 -3521.905,E2 -3521.905} C_VEL
LIN {X 0,Y 545.085,Z 516.589,A -85,B 0,C 180,E1 -3524.945,E2 -3524.945} C_VEL
LIN {X 0,Y 545.072,Z 516.582,A -85,B 0,C 180,E1 -3528.027,E2 -3528.027} C_VEL
LIN {X 0,Y 545.095,Z 516.58,A -85,B 0,C 180,E1 -3530.373,E2 -3530.373} C_VEL
LIN {X 0,Y 545.08,Z 516.585,A -85,B 0,C 180,E1 -3533.56,E2 -3533.56} C_VEL
LIN {X 0,Y 545.08,Z 516.582,A -85,B 0,C 180,E1 -3536.001,E2 -3536.001} C_VEL
LIN {X 0,Y 545.09,Z 516.583,A -85,B 0,C 180,E1 -3538.749,E2 -3538.749} C_VEL
LIN {X 0,Y 545.059,Z 516.587,A -85,B 0,C 180,E1 -3541.68,E2 -3541.68} C_VEL
LIN {X 0,Y 545.063,Z 516.584,A -85,B 0,C 180,E1 -3544.565,E2 -3544.565} C_VEL
LIN {X 0,Y 545.039,Z 516.597,A -85,B 0,C 180,E1 -3547.305,E2 -3547.305} C_VEL
LIN {X 0,Y 545.074,Z 516.583,A -85,B 0,C 180,E1 -3550.143,E2 -3550.143} C_VEL
LIN {X 0,Y 545.089,Z 516.586,A -85,B 0,C 180,E1 -3553.107,E2 -3553.107} C_VEL
LIN {X 0,Y 545.053,Z 516.585,A -85,B 0,C 180,E1 -3556.227,E2 -3556.227} C_VEL
LIN {X 0,Y 545.094,Z 516.582,A -85,B 0,C 180,E1 -3558.887,E2 -3558.887} C_VEL
LIN {X 0,Y 545.056,Z 516.589,A -85,B 0,C 180,E1 -3561.764,E2 -3561.764} C_VEL
LIN {X 0,Y 545.042,Z 516.586,A -85,B 0,C 180,E1 -3564.532,E2 -3564.532} C_VEL
LIN {X 0,Y 545.085,Z 516.586,A -85,B 0,C 180,E1 -3567.213,E2 -3567.213} C_VEL
LIN {X 0,Y 545.068,Z 516.588,A -85,B 0,C 180,E1 -3569.811,E2 -3569.811} C_VEL
LIN {X 0,Y 545.085,Z 516.581,A -85,B 0,C 180,E1 -3572.344,E2 -3572.344} C_VEL
LIN {X 0,Y 545.122,Z 516.577,A -85,B 0,C 180,E1 -3574.821,E2 -3574.821} C_VEL
LIN {X 0,Y 545.041,Z 516.591,A -85,B 0,C 180,E1 -3577.243,E2 -3577.243} C_VEL
LIN {X 0,Y 545.121,Z 516.577,A -85,B 0,C 180,E1 -3580.415,E2 -3580.415} C_VEL
LIN {X 0,Y 545.079,Z 516.589,A -85,B 0,C 180,E1 -3583.522,E2 -3583.522} C_VEL
LIN {X 0,Y 545.1,Z 516.587,A -85,B 0,C 180,E1 -3585.82,E2 -3585.82} C_VEL
LIN {X 0,Y 545.123,Z 516.576,A -85,B 0,C 180,E1 -3588.85,E2 -3588.85} C_VEL
LIN {X 0,Y 545.134,Z 516.583,A -85,B 0,C 180,E1 -3591.848,E2 -3591.848} C_VEL
LIN {X 0,Y 545.209,Z 516.565,A -85,B 0,C 180,E1 -3594.823,E2 -3594.823} C_VEL
LIN {X 0,Y 545.2,Z 516.576,A -85,B 0,C 180,E1 -3597.784,E2 -3597.784} C_VEL
LIN {X 0,Y 545.218,Z 516.564,A -85,B 0,C 180,E1 -3600.739,E2 -3600.739} C_VEL
LIN {X 0,Y 545.177,Z 516.569,A -85,B 0,C 180,E1 -3602.956,E2 -3602.956} C_VEL
LIN {X 0,Y 545.177,Z 516.579,A -85,B 0,C 180,E1 -3605.92,E2 -3605.92} C_VEL
LIN {X 0,Y 545.117,Z 516.577,A -85,B 0,C 180,E1 -3608.9,E2 -3608.9} C_VEL
LIN {X 0,Y 545.142,Z 516.583,A -85,B 0,C 180,E1 -3611.904,E2 -3611.904} C_VEL
LIN {X 0,Y 545.093,Z 516.58,A -85,B 0,C 180,E1 -3614.944,E2 -3614.944} C_VEL
LIN {X 0,Y 545.078,Z 516.592,A -85,B 0,C 180,E1 -3618.026,E2 -3618.026} C_VEL
LIN {X 0,Y 545.1,Z 516.584,A -85,B 0,C 180,E1 -3620.372,E2 -3620.372} C_VEL
LIN {X 0,Y 545.086,Z 516.583,A -85,B 0,C 180,E1 -3623.559,E2 -3623.559} C_VEL
LIN {X 0,Y 545.085,Z 516.589,A -85,B 0,C 180,E1 -3626.001,E2 -3626.001} C_VEL
LIN {X 0,Y 545.097,Z 516.581,A -85,B 0,C 180,E1 -3628.748,E2 -3628.748} C_VEL
LIN {X 0,Y 545.065,Z 516.586,A -85,B 0,C 180,E1 -3631.679,E2 -3631.679} C_VEL
LIN {X 0,Y 545.072,Z 516.586,A -85,B 0,C 180,E1 -3634.564,E2 -3634.564} C_VEL
LIN {X 0,Y 545.044,Z 516.586,A -85,B 0,C 180,E1 -3637.304,E2 -3637.304} C_VEL
LIN {X 0,Y 545.073,Z 516.591,A -85,B 0,C 180,E1 -3640.142,E2 -3640.142} C_VEL
LIN {X 0,Y 545.045,Z 516.589,A -85,B 0,C 180,E1 -3642.694,E2 -3642.694} C_VEL
LIN {X 0,Y 545.04,Z 516.587,A -85,B 0,C 180,E1 -3645.17,E2 -3645.17} C_VEL
LIN {X 0,Y 545.085,Z 516.584,A -85,B 0,C 180,E1 -3647.897,E2 -3647.897} C_VEL
LIN {X 0,Y 545.086,Z 516.583,A -85,B 0,C 180,E1 -3650.818,E2 -3650.818} C_VEL
LIN {X 0,Y 545.049,Z 516.586,A -85,B 0,C 180,E1 -3653.619,E2 -3653.619} C_VEL
LIN {X 0,Y 545.073,Z 516.591,A -85,B 0,C 180,E1 -3656.328,E2 -3656.328} C_VEL
LIN {X 0,Y 545.073,Z 516.586,A -85,B 0,C 180,E1 -3658.952,E2 -3658.952} C_VEL
LIN {X 0,Y 545.109,Z 516.579,A -85,B 0,C 180,E1 -3661.507,E2 -3661.507} C_VEL
LIN {X 0,Y 545.101,Z 516.589,A -85,B 0,C 180,E1 -3664.491,E2 -3664.491} C_VEL
LIN {X 0,Y 545.071,Z 516.651,A -85,B 0,C 180,E1 -3666.284,E2 -3666.284} C_VEL
LIN {X 0,Y 546.296,Z 523.851,A -85,B 0,C 180,E1 -3667.473,E2 -3667.473} C_VEL
LIN {X 0,Y 545.897,Z 543.101,A -85,B 0,C 180,E1 -3670.443,E2 -3670.443} C_VEL
LIN {X 0,Y 545.609,Z 559.572,A -85,B 0,C 180,E1 -3672.959,E2 -3672.959} C_VEL
LIN {X 0,Y 545.376,Z 575.906,A -85,B 0,C 180,E1 -3675.44,E2 -3675.44} C_VEL
LIN {X 0,Y 546.57,Z 584.818,A -85,B 0,C 180,E1 -3675.594,E2 -3675.594} C_VEL
LIN {X 0,Y 546.211,Z 683.899,A -85,B 0,C 180,E1 -3676.915,E2 -3676.915} C_VEL
LIN {X 0,Y 546.063,Z 697.186,A -85,B 0,C 180,E1 -3677.243,E2 -3677.243} C_VEL
LIN {X 0,Y 545.91,Z 709.347,A -85,B 0,C 180,E1 -3677.688,E2 -3677.688} C_VEL
LIN {X 0,Y 545.708,Z 720.387,A -85,B 0,C 180,E1 -3678.227,E2 -3678.227} C_VEL
LIN {X 0,Y 545.539,Z 731.891,A -85,B 0,C 180,E1 -3678.951,E2 -3678.951} C_VEL
LIN {X 0,Y 545.284,Z 742.526,A -85,B 0,C 180,E1 -3679.791,E2 -3679.791} C_VEL
LIN {X 0,Y 545.085,Z 752.104,A -85,B 0,C 180,E1 -3680.724,E2 -3680.724} C_VEL
LIN {X 0,Y 544.977,Z 759.953,A -85,B 0,C 180,E1 -3681.657,E2 -3681.657} C_VEL
LIN {X 0,Y 544.824,Z 767.615,A -85,B 0,C 180,E1 -3682.774,E2 -3682.774} C_VEL
LIN {X 0,Y 544.777,Z 774.675,A -85,B 0,C 180,E1 -3684.075,E2 -3684.075} C_VEL
LIN {X 0,Y 544.629,Z 779.369,A -85,B 0,C 180,E1 -3685.188,E2 -3685.188} C_VEL
LIN {X 0,Y 544.669,Z 782.955,A -85,B 0,C 180,E1 -3686.3,E2 -3686.3} C_VEL
LIN {X 0,Y 544.651,Z 784.805,A -85,B 0,C 180,E1 -3687.04,E2 -3687.04} C_VEL
LIN {X 0,Y 544.546,Z 787.182,A -85,B 0,C 180,E1 -3688.52,E2 -3688.52} C_VEL
LIN {X 0,Y 544.541,Z 788,A -85,B 0,C 180,E1 -3689.999,E2 -3689.999} C_VEL
LIN {X 0,Y 544.546,Z 787.186,A -85,B 0,C 180,E1 -3691.478,E2 -3691.478} C_VEL
LIN {X 0,Y 544.65,Z 784.812,A -85,B 0,C 180,E1 -3692.958,E2 -3692.958} C_VEL
LIN {X 0,Y 544.683,Z 781.899,A -85,B 0,C 180,E1 -3694.068,E2 -3694.068} C_VEL
LIN {X 0,Y 544.654,Z 777.953,A -85,B 0,C 180,E1 -3695.181,E2 -3695.181} C_VEL
LIN {X 0,Y 544.728,Z 772.656,A -85,B 0,C 180,E1 -3696.337,E2 -3696.337} C_VEL
LIN {X 0,Y 544.859,Z 765.244,A -85,B 0,C 180,E1 -3697.596,E2 -3697.596} C_VEL
LIN {X 0,Y 545.028,Z 757,A -85,B 0,C 180,E1 -3698.713,E2 -3698.713} C_VEL
LIN {X 0,Y 545.201,Z 748.551,A -85,B 0,C 180,E1 -3699.646,E2 -3699.646} C_VEL
LIN {X 0,Y 545.391,Z 738.108,A -85,B 0,C 180,E1 -3700.58,E2 -3700.58} C_VEL
LIN {X 0,Y 545.614,Z 726.371,A -85,B 0,C 180,E1 -3701.42,E2 -3701.42} C_VEL
LIN {X 0,Y 545.848,Z 714.513,A -85,B 0,C 180,E1 -3702.076,E2 -3702.076} C_VEL
LIN {X 0,Y 546.004,Z 702.198,A -85,B 0,C 180,E1 -3702.591,E2 -3702.591} C_VEL
LIN {X 0,Y 546.138,Z 689.562,A -85,B 0,C 180,E1 -3702.966,E2 -3702.966} C_VEL
LIN {X 0,Y 546.267,Z 676.399,A -85,B 0,C 180,E1 -3703.2,E2 -3703.2} C_VEL
LIN {X 0,Y 546.437,Z 582.737,A -85,B 0,C 180,E1 -3704.437,E2 -3704.437} C_VEL
LIN {X 0,Y 545.377,Z 575.881,A -85,B 0,C 180,E1 -3704.564,E2 -3704.564} C_VEL
LIN {X 0,Y 545.693,Z 554.939,A -85,B 0,C 180,E1 -3707.75,E2 -3707.75} C_VEL
LIN {X 0,Y 546.057,Z 535.469,A -85,B 0,C 180,E1 -3710.727,E2 -3710.727} C_VEL
LIN {X 0,Y 546.249,Z 522.7,A -85,B 0,C 180,E1 -3712.703,E2 -3712.703} C_VEL
LIN {X 0,Y 545.092,Z 516.59,A -85,B 0,C 180,E1 -3713.734,E2 -3713.734} C_VEL
LIN {X 0,Y 545.078,Z 516.587,A -85,B 0,C 180,E1 -3715.999,E2 -3715.999} C_VEL
LIN {X 0,Y 545.087,Z 516.585,A -85,B 0,C 180,E1 -3718.747,E2 -3718.747} C_VEL
LIN {X 0,Y 545.076,Z 516.59,A -85,B 0,C 180,E1 -3721.681,E2 -3721.681} C_VEL
LIN {X 0,Y 545.073,Z 516.583,A -85,B 0,C 180,E1 -3724.562,E2 -3724.562} C_VEL
LIN {X 0,Y 545.036,Z 516.596,A -85,B 0,C 180,E1 -3727.302,E2 -3727.302} C_VEL
LIN {X 0,Y 545.072,Z 516.585,A -85,B 0,C 180,E1 -3730.14,E2 -3730.14} C_VEL
LIN {X 0,Y 545.081,Z 516.587,A -85,B 0,C 180,E1 -3733.104,E2 -3733.104} C_VEL
LIN {X 0,Y 545.06,Z 516.586,A -85,B 0,C 180,E1 -3736.223,E2 -3736.223} C_VEL
LIN {X 0,Y 545.094,Z 516.583,A -85,B 0,C 180,E1 -3738.886,E2 -3738.886} C_VEL
LIN {X 0,Y 545.047,Z 516.59,A -85,B 0,C 180,E1 -3741.762,E2 -3741.762} C_VEL
LIN {X 0,Y 545.059,Z 516.585,A -85,B 0,C 180,E1 -3744.533,E2 -3744.533} C_VEL
LIN {X 0,Y 545.075,Z 516.588,A -85,B 0,C 180,E1 -3747.212,E2 -3747.212} C_VEL
LIN {X 0,Y 545.093,Z 516.585,A -85,B 0,C 180,E1 -3749.812,E2 -3749.812} C_VEL
LIN {X 0,Y 545.093,Z 516.581,A -85,B 0,C 180,E1 -3752.824,E2 -3752.824} C_VEL
LIN {X 0,Y 545.044,Z 516.592,A -85,B 0,C 180,E1 -3755.63,E2 -3755.63} C_VEL
LIN {X 0,Y 545.06,Z 516.586,A -85,B 0,C 180,E1 -3758.836,E2 -3758.836} C_VEL
LIN {X 0,Y 545.076,Z 516.586,A -85,B 0,C 180,E1 -3761.195,E2 -3761.195} C_VEL
LIN {X 0,Y 545.068,Z 516.59,A -85,B 0,C 180,E1 -3763.521,E2 -3763.521} C_VEL
LIN {X 0,Y 545.085,Z 516.585,A -85,B 0,C 180,E1 -3765.819,E2 -3765.819} C_VEL
LIN {X 0,Y 545.122,Z 516.577,A -85,B 0,C 180,E1 -3768.849,E2 -3768.849} C_VEL
LIN {X 0,Y 545.124,Z 516.579,A -85,B 0,C 180,E1 -3771.847,E2 -3771.847} C_VEL
LIN {X 0,Y 545.2,Z 516.569,A -85,B 0,C 180,E1 -3774.823,E2 -3774.823} C_VEL
LIN {X 0,Y 545.186,Z 516.572,A -85,B 0,C 180,E1 -3777.783,E2 -3777.783} C_VEL
LIN {X 0,Y 545.206,Z 516.568,A -85,B 0,C 180,E1 -3780.738,E2 -3780.738} C_VEL
LIN {X 0,Y 545.168,Z 516.574,A -85,B 0,C 180,E1 -3782.955,E2 -3782.955} C_VEL
LIN {X 0,Y 545.162,Z 516.575,A -85,B 0,C 180,E1 -3785.919,E2 -3785.919} C_VEL
LIN {X 0,Y 545.118,Z 516.58,A -85,B 0,C 180,E1 -3788.9,E2 -3788.9} C_VEL
LIN {X 0,Y 545.124,Z 516.58,A -85,B 0,C 180,E1 -3791.904,E2 -3791.904} C_VEL
LIN {X 0,Y 545.074,Z 516.587,A -85,B 0,C 180,E1 -3794.943,E2 -3794.943} C_VEL
LIN {X 0,Y 545.072,Z 516.586,A -85,B 0,C 180,E1 -3798.026,E2 -3798.026} C_VEL
LIN {X 0,Y 545.087,Z 516.582,A -85,B 0,C 180,E1 -3800.372,E2 -3800.372} C_VEL
LIN {X 0,Y 545.08,Z 516.591,A -85,B 0,C 180,E1 -3803.559,E2 -3803.559} C_VEL
LIN {X 0,Y 545.078,Z 516.586,A -85,B 0,C 180,E1 -3806,E2 -3806} C_VEL
LIN {X 0,Y 545.082,Z 516.587,A -85,B 0,C 180,E1 -3808.75,E2 -3808.75} C_VEL
LIN {X 0,Y 545.098,Z 516.631,A -85,B 0,C 180,E1 -3809.814,E2 -3809.814} C_VEL
LIN {X 0,Y 545.645,Z 520.717,A -85,B 0,C 180,E1 -3810.612,E2 -3810.612} C_VEL
LIN {X 0,Y 545.33,Z 537.062,A -85,B 0,C 180,E1 -3813.653,E2 -3813.653} C_VEL
LIN {X 0,Y 545.205,Z 545.046,A -85,B 0,C 180,E1 -3815.109,E2 -3815.109} C_VEL
LIN {X 0,Y 544.818,Z 546.858,A -85,B 0,C 180,E1 -3815.31,E2 -3815.31} C_VEL
LIN {X 0,Y 543.598,Z 550.02,A -85,B 0,C 180,E1 -3815.457,E2 -3815.457} C_VEL
LIN {X 0,Y 541.652,Z 554.565,A -85,B 0,C 180,E1 -3815.502,E2 -3815.502} C_VEL
LIN {X 0,Y 539.99,Z 560.531,A -85,B 0,C 180,E1 -3815.531,E2 -3815.531} C_VEL
LIN {X 0,Y 539.548,Z 566.992,A -85,B 0,C 180,E1 -3815.604,E2 -3815.604} C_VEL
LIN {X 0,Y 539.605,Z 575.669,A -85,B 0,C 180,E1 -3815.73,E2 -3815.73} C_VEL
LIN {X 0,Y 539.286,Z 654.726,A -85,B 0,C 180,E1 -3816.805,E2 -3816.805} C_VEL
LIN {X 0,Y 539.098,Z 668.519,A -85,B 0,C 180,E1 -3817.162,E2 -3817.162} C_VEL
LIN {X 0,Y 538.914,Z 681.157,A -85,B 0,C 180,E1 -3817.651,E2 -3817.651} C_VEL
LIN {X 0,Y 538.69,Z 693.211,A -85,B 0,C 180,E1 -3818.283,E2 -3818.283} C_VEL
LIN {X 0,Y 538.435,Z 704.428,A -85,B 0,C 180,E1 -3819.034,E2 -3819.034} C_VEL
LIN {X 0,Y 538.244,Z 714.685,A -85,B 0,C 180,E1 -3819.899,E2 -3819.899} C_VEL
LIN {X 0,Y 538.027,Z 724.355,A -85,B 0,C 180,E1 -3820.901,E2 -3820.901} C_VEL
LIN {X 0,Y 537.835,Z 733.282,A -85,B 0,C 180,E1 -3822.055,E2 -3822.055} C_VEL
LIN {X 0,Y 537.687,Z 740.037,A -85,B 0,C 180,E1 -3823.138,E2 -3823.138} C_VEL
LIN {X 0,Y 537.647,Z 744.642,A -85,B 0,C 180,E1 -3824.034,E2 -3824.034} C_VEL
LIN {X 0,Y 537.599,Z 749.098,A -85,B 0,C 180,E1 -3825.097,E2 -3825.097} C_VEL
LIN {X 0,Y 537.525,Z 752.521,A -85,B 0,C 180,E1 -3826.137,E2 -3826.137} C_VEL
LIN {X 0,Y 537.497,Z 755.056,A -85,B 0,C 180,E1 -3827.164,E2 -3827.164} C_VEL
LIN {X 0,Y 537.488,Z 756.768,A -85,B 0,C 180,E1 -3828.185,E2 -3828.185} C_VEL
LIN {X 0,Y 537.452,Z 757.803,A -85,B 0,C 180,E1 -3829.326,E2 -3829.326} C_VEL
LIN {X 0,Y 537.421,Z 757.913,A -85,B 0,C 180,E1 -3830.493,E2 -3830.493} C_VEL
LIN {X 0,Y 537.423,Z 757.037,A -85,B 0,C 180,E1 -3831.686,E2 -3831.686} C_VEL
LIN {X 0,Y 537.474,Z 754.84,A -85,B 0,C 180,E1 -3833.025,E2 -3833.025} C_VEL
LIN {X 0,Y 537.546,Z 751.935,A -85,B 0,C 180,E1 -3834.154,E2 -3834.154} C_VEL
LIN {X 0,Y 537.532,Z 747.286,A -85,B 0,C 180,E1 -3835.456,E2 -3835.456} C_VEL
LIN {X 0,Y 537.692,Z 741.035,A -85,B 0,C 180,E1 -3836.774,E2 -3836.774} C_VEL
LIN {X 0,Y 537.798,Z 734.183,A -85,B 0,C 180,E1 -3837.903,E2 -3837.903} C_VEL
LIN {X 0,Y 537.987,Z 726.47,A -85,B 0,C 180,E1 -3838.937,E2 -3838.937} C_VEL
LIN {X 0,Y 538.144,Z 717.498,A -85,B 0,C 180,E1 -3839.924,E2 -3839.924} C_VEL
LIN {X 0,Y 538.395,Z 706.843,A -85,B 0,C 180,E1 -3840.866,E2 -3840.866} C_VEL
LIN {X 0,Y 538.629,Z 695.549,A -85,B 0,C 180,E1 -3841.667,E2 -3841.667} C_VEL
LIN {X 0,Y 538.852,Z 684.641,A -85,B 0,C 180,E1 -3842.275,E2 -3842.275} C_VEL
LIN {X 0,Y 539.038,Z 672.586,A -85,B 0,C 180,E1 -3842.788,E2 -3842.788} C_VEL
LIN {X 0,Y 539.258,Z 659.691,A -85,B 0,C 180,E1 -3843.177,E2 -3843.177} C_VEL
LIN {X 0,Y 539.378,Z 646.229,A -85,B 0,C 180,E1 -3843.418,E2 -3843.418} C_VEL
LIN {X 0,Y 539.644,Z 555.864,A -85,B 0,C 180,E1 -3844.626,E2 -3844.626} C_VEL
LIN {X 0,Y 538.158,Z 547.239,A -85,B 0,C 180,E1 -3844.784,E2 -3844.784} C_VEL
LIN {X 0,Y 538.447,Z 531.305,A -85,B 0,C 180,E1 -3847.759,E2 -3847.759} C_VEL
LIN {X 0,Y 538.578,Z 520.711,A -85,B 0,C 180,E1 -3849.771,E2 -3849.771} C_VEL
LIN {X 0,Y 538.076,Z 517.464,A -85,B 0,C 180,E1 -3850.447,E2 -3850.447} C_VEL
LIN {X 0,Y 538.021,Z 517.465,A -85,B 0,C 180,E1 -3853.3,E2 -3853.3} C_VEL
LIN {X 0,Y 538.06,Z 517.458,A -85,B 0,C 180,E1 -3855.632,E2 -3855.632} C_VEL
LIN {X 0,Y 538.073,Z 517.463,A -85,B 0,C 180,E1 -3858.703,E2 -3858.703} C_VEL
LIN {X 0,Y 538.083,Z 517.453,A -85,B 0,C 180,E1 -3861.741,E2 -3861.741} C_VEL
LIN {X 0,Y 538.161,Z 517.452,A -85,B 0,C 180,E1 -3864.756,E2 -3864.756} C_VEL
LIN {X 0,Y 538.167,Z 517.443,A -85,B 0,C 180,E1 -3867.756,E2 -3867.756} C_VEL
LIN {X 0,Y 538.181,Z 517.448,A -85,B 0,C 180,E1 -3870.749,E2 -3870.749} C_VEL
LIN {X 0,Y 538.137,Z 517.456,A -85,B 0,C 180,E1 -3872.996,E2 -3872.996} C_VEL
LIN {X 0,Y 538.118,Z 517.449,A -85,B 0,C 180,E1 -3875.998,E2 -3875.998} C_VEL
LIN {X 0,Y 538.067,Z 517.465,A -85,B 0,C 180,E1 -3879.019,E2 -3879.019} C_VEL
LIN {X 0,Y 538.083,Z 517.453,A -85,B 0,C 180,E1 -3882.064,E2 -3882.064} C_VEL
LIN {X 0,Y 538.045,Z 517.467,A -85,B 0,C 180,E1 -3885.145,E2 -3885.145} C_VEL
LIN {X 0,Y 538.027,Z 517.46,A -85,B 0,C 180,E1 -3888.271,E2 -3888.271} C_VEL
LIN {X 0,Y 538.04,Z 517.461,A -85,B 0,C 180,E1 -3890.652,E2 -3890.652} C_VEL
LIN {X 0,Y 538.003,Z 517.464,A -85,B 0,C 180,E1 -3893.889,E2 -3893.889} C_VEL
LIN {X 0,Y 538.042,Z 517.458,A -85,B 0,C 180,E1 -3896.368,E2 -3896.368} C_VEL
LIN {X 0,Y 538.032,Z 517.465,A -85,B 0,C 180,E1 -3898.934,E2 -3898.934} C_VEL
LIN {X 0,Y 538.012,Z 517.463,A -85,B 0,C 180,E1 -3901.888,E2 -3901.888} C_VEL
LIN {X 0,Y 538.013,Z 517.463,A -85,B 0,C 180,E1 -3904.619,E2 -3904.619} C_VEL
LIN {X 0,Y 538.007,Z 517.471,A -85,B 0,C 180,E1 -3907.171,E2 -3907.171} C_VEL
LIN {X 0,Y 538.029,Z 517.463,A -85,B 0,C 180,E1 -3909.797,E2 -3909.797} C_VEL
LIN {X 0,Y 538.026,Z 517.462,A -85,B 0,C 180,E1 -3912.786,E2 -3912.786} C_VEL
LIN {X 0,Y 538.035,Z 517.465,A -85,B 0,C 180,E1 -3915.141,E2 -3915.141} C_VEL
LIN {X 0,Y 538.037,Z 517.459,A -85,B 0,C 180,E1 -3918.228,E2 -3918.228} C_VEL
LIN {X 0,Y 538.018,Z 517.467,A -85,B 0,C 180,E1 -3921.171,E2 -3921.171} C_VEL
LIN {X 0,Y 537.998,Z 517.465,A -85,B 0,C 180,E1 -3924.089,E2 -3924.089} C_VEL
LIN {X 0,Y 538.035,Z 517.46,A -85,B 0,C 180,E1 -3926.728,E2 -3926.728} C_VEL
LIN {X 0,Y 538.03,Z 517.469,A -85,B 0,C 180,E1 -3929.557,E2 -3929.557} C_VEL
LIN {X 0,Y 538.044,Z 517.462,A -85,B 0,C 180,E1 -3931.951,E2 -3931.951} C_VEL
LIN {X 0,Y 538.076,Z 517.454,A -85,B 0,C 180,E1 -3934.468,E2 -3934.468} C_VEL
LIN {X 0,Y 537.998,Z 517.471,A -85,B 0,C 180,E1 -3937.739,E2 -3937.739} C_VEL
LIN {X 0,Y 538.085,Z 517.455,A -85,B 0,C 180,E1 -3940.149,E2 -3940.149} C_VEL
LIN {X 0,Y 538.025,Z 517.465,A -85,B 0,C 180,E1 -3943.299,E2 -3943.299} C_VEL
LIN {X 0,Y 538.069,Z 517.464,A -85,B 0,C 180,E1 -3945.631,E2 -3945.631} C_VEL
LIN {X 0,Y 538.083,Z 517.453,A -85,B 0,C 180,E1 -3948.702,E2 -3948.702} C_VEL
LIN {X 0,Y 538.09,Z 517.463,A -85,B 0,C 180,E1 -3951.74,E2 -3951.74} C_VEL
LIN {X 0,Y 538.167,Z 517.443,A -85,B 0,C 180,E1 -3954.755,E2 -3954.755} C_VEL
LIN {X 0,Y 538.172,Z 517.451,A -85,B 0,C 180,E1 -3957.755,E2 -3957.755} C_VEL
LIN {X 0,Y 538.189,Z 517.44,A -85,B 0,C 180,E1 -3960.749,E2 -3960.749} C_VEL
LIN {X 0,Y 538.144,Z 517.446,A -85,B 0,C 180,E1 -3962.995,E2 -3962.995} C_VEL
LIN {X 0,Y 538.13,Z 517.455,A -85,B 0,C 180,E1 -3965.998,E2 -3965.998} C_VEL
LIN {X 0,Y 538.067,Z 517.455,A -85,B 0,C 180,E1 -3969.018,E2 -3969.018} C_VEL
LIN {X 0,Y 538.09,Z 517.46,A -85,B 0,C 180,E1 -3972.063,E2 -3972.063} C_VEL
LIN {X 0,Y 538.053,Z 517.457,A -85,B 0,C 180,E1 -3975.144,E2 -3975.144} C_VEL
LIN {X 0,Y 538.033,Z 517.465,A -85,B 0,C 180,E1 -3978.271,E2 -3978.271} C_VEL
LIN {X 0,Y 538.045,Z 517.459,A -85,B 0,C 180,E1 -3980.651,E2 -3980.651} C_VEL
LIN {X 0,Y 538.01,Z 517.469,A -85,B 0,C 180,E1 -3983.888,E2 -3983.888} C_VEL
LIN {X 0,Y 538.047,Z 517.463,A -85,B 0,C 180,E1 -3986.367,E2 -3986.367} C_VEL
LIN {X 0,Y 538.038,Z 517.459,A -85,B 0,C 180,E1 -3988.933,E2 -3988.933} C_VEL
LIN {X 0,Y 538.017,Z 517.467,A -85,B 0,C 180,E1 -3991.887,E2 -3991.887} C_VEL
LIN {X 0,Y 538.023,Z 517.464,A -85,B 0,C 180,E1 -3994.618,E2 -3994.618} C_VEL
LIN {X 0,Y 538.013,Z 517.462,A -85,B 0,C 180,E1 -3997.17,E2 -3997.17} C_VEL
LIN {X 0,Y 538.03,Z 517.463,A -85,B 0,C 180,E1 -3999.797,E2 -3999.797} C_VEL
LIN {X 0,Y 537.994,Z 517.466,A -85,B 0,C 180,E1 -4002.789,E2 -4002.789} C_VEL
LIN {X 0,Y 538.01,Z 517.462,A -85,B 0,C 180,E1 -4005.137,E2 -4005.137} C_VEL
LIN {X 0,Y 538.038,Z 517.467,A -85,B 0,C 180,E1 -4008.226,E2 -4008.226} C_VEL
LIN {X 0,Y 538.019,Z 517.461,A -85,B 0,C 180,E1 -4011.169,E2 -4011.169} C_VEL
LIN {X 0,Y 538.001,Z 517.469,A -85,B 0,C 180,E1 -4014.088,E2 -4014.088} C_VEL
LIN {X 0,Y 538.037,Z 517.463,A -85,B 0,C 180,E1 -4016.727,E2 -4016.727} C_VEL
LIN {X 0,Y 538.033,Z 517.461,A -85,B 0,C 180,E1 -4019.556,E2 -4019.556} C_VEL
LIN {X 0,Y 538.064,Z 517.464,A -85,B 0,C 180,E1 -4022.647,E2 -4022.647} C_VEL
LIN {X 0,Y 538.055,Z 517.462,A -85,B 0,C 180,E1 -4025.292,E2 -4025.292} C_VEL
LIN {X 0,Y 538.049,Z 517.493,A -85,B 0,C 180,E1 -4026.113,E2 -4026.113} C_VEL
LIN {X 0,Y 539.366,Z 525.363,A -85,B 0,C 180,E1 -4027.434,E2 -4027.434} C_VEL
LIN {X 0,Y 538.901,Z 545.484,A -85,B 0,C 180,E1 -4030.575,E2 -4030.575} C_VEL
LIN {X 0,Y 538.543,Z 563.283,A -85,B 0,C 180,E1 -4033.315,E2 -4033.315} C_VEL
LIN {X 0,Y 538.368,Z 575.923,A -85,B 0,C 180,E1 -4035.248,E2 -4035.248} C_VEL
LIN {X 0,Y 539.687,Z 584.965,A -85,B 0,C 180,E1 -4035.408,E2 -4035.408} C_VEL
LIN {X 0,Y 539.322,Z 683.898,A -85,B 0,C 180,E1 -4036.745,E2 -4036.745} C_VEL
LIN {X 0,Y 539.136,Z 697.185,A -85,B 0,C 180,E1 -4037.076,E2 -4037.076} C_VEL
LIN {X 0,Y 538.956,Z 709.346,A -85,B 0,C 180,E1 -4037.526,E2 -4037.526} C_VEL
LIN {X 0,Y 538.731,Z 721.697,A -85,B 0,C 180,E1 -4038.148,E2 -4038.148} C_VEL
LIN {X 0,Y 538.544,Z 733.181,A -85,B 0,C 180,E1 -4038.901,E2 -4038.901} C_VEL
LIN {X 0,Y 538.259,Z 743.594,A -85,B 0,C 180,E1 -4039.752,E2 -4039.752} C_VEL
LIN {X 0,Y 538.068,Z 752.104,A -85,B 0,C 180,E1 -4040.602,E2 -4040.602} C_VEL
LIN {X 0,Y 537.92,Z 759.953,A -85,B 0,C 180,E1 -4041.547,E2 -4041.547} C_VEL
LIN {X 0,Y 537.756,Z 767.616,A -85,B 0,C 180,E1 -4042.678,E2 -4042.678} C_VEL
LIN {X 0,Y 537.694,Z 774.674,A -85,B 0,C 180,E1 -4043.997,E2 -4043.997} C_VEL
LIN {X 0,Y 537.541,Z 779.369,A -85,B 0,C 180,E1 -4045.124,E2 -4045.124} C_VEL
LIN {X 0,Y 537.591,Z 782.955,A -85,B 0,C 180,E1 -4046.251,E2 -4046.251} C_VEL
LIN {X 0,Y 537.551,Z 784.805,A -85,B 0,C 180,E1 -4047.001,E2 -4047.001} C_VEL
LIN {X 0,Y 537.451,Z 787.182,A -85,B 0,C 180,E1 -4048.5,E2 -4048.5} C_VEL
LIN {X 0,Y 537.442,Z 788,A -85,B 0,C 180,E1 -4049.999,E2 -4049.999} C_VEL
LIN {X 0,Y 537.451,Z 787.185,A -85,B 0,C 180,E1 -4051.498,E2 -4051.498} C_VEL
LIN {X 0,Y 537.551,Z 784.812,A -85,B 0,C 180,E1 -4052.997,E2 -4052.997} C_VEL
LIN {X 0,Y 537.603,Z 781.898,A -85,B 0,C 180,E1 -4054.122,E2 -4054.122} C_VEL
LIN {X 0,Y 537.587,Z 777.952,A -85,B 0,C 180,E1 -4055.25,E2 -4055.25} C_VEL
LIN {X 0,Y 537.642,Z 773.136,A -85,B 0,C 180,E1 -4056.324,E2 -4056.324} C_VEL
LIN {X 0,Y 537.79,Z 766.474,A -85,B 0,C 180,E1 -4057.508,E2 -4057.508} C_VEL
LIN {X 0,Y 537.972,Z 758.486,A -85,B 0,C 180,E1 -4058.639,E2 -4058.639} C_VEL
LIN {X 0,Y 538.142,Z 750.344,A -85,B 0,C 180,E1 -4059.584,E2 -4059.584} C_VEL
LIN {X 0,Y 538.352,Z 740.411,A -85,B 0,C 180,E1 -4060.53,E2 -4060.53} C_VEL
LIN {X 0,Y 538.583,Z 730.608,A -85,B 0,C 180,E1 -4061.287,E2 -4061.287} C_VEL
LIN {X 0,Y 538.803,Z 719.724,A -85,B 0,C 180,E1 -4061.962,E2 -4061.962} C_VEL
LIN {X 0,Y 539.005,Z 707.13,A -85,B 0,C 180,E1 -4062.566,E2 -4062.566} C_VEL
LIN {X 0,Y 539.191,Z 694.131,A -85,B 0,C 180,E1 -4063.016,E2 -4063.016} C_VEL
LIN {X 0,Y 539.348,Z 681.179,A -85,B 0,C 180,E1 -4063.3,E2 -4063.3} C_VEL
LIN {X 0,Y 539.582,Z 583.488,A -85,B 0,C 180,E1 -4064.614,E2 -4064.614} C_VEL
LIN {X 0,Y 538.391,Z 575.898,A -85,B 0,C 180,E1 -4064.755,E2 -4064.755} C_VEL
LIN {X 0,Y 538.765,Z 554.12,A -85,B 0,C 180,E1 -4068.088,E2 -4068.088} C_VEL
LIN {X 0,Y 539.126,Z 533.991,A -85,B 0,C 180,E1 -4071.206,E2 -4071.206} C_VEL
LIN {X 0,Y 539.266,Z 523.775,A -85,B 0,C 180,E1 -4072.811,E2 -4072.811} C_VEL
LIN {X 0,Y 538.041,Z 517.467,A -85,B 0,C 180,E1 -4073.885,E2 -4073.885} C_VEL
LIN {X 0,Y 538.041,Z 517.462,A -85,B 0,C 180,E1 -4076.365,E2 -4076.365} C_VEL
LIN {X 0,Y 538.029,Z 517.466,A -85,B 0,C 180,E1 -4078.932,E2 -4078.932} C_VEL
LIN {X 0,Y 538.025,Z 517.466,A -85,B 0,C 180,E1 -4081.889,E2 -4081.889} C_VEL
LIN {X 0,Y 538.023,Z 517.462,A -85,B 0,C 180,E1 -4084.619,E2 -4084.619} C_VEL
LIN {X 0,Y 538.003,Z 517.47,A -85,B 0,C 180,E1 -4087.169,E2 -4087.169} C_VEL
LIN {X 0,Y 538.029,Z 517.466,A -85,B 0,C 180,E1 -4089.795,E2 -4089.795} C_VEL
LIN {X 0,Y 538.018,Z 517.464,A -85,B 0,C 180,E1 -4092.784,E2 -4092.784} C_VEL
LIN {X 0,Y 538.023,Z 517.465,A -85,B 0,C 180,E1 -4095.924,E2 -4095.924} C_VEL
LIN {X 0,Y 538.072,Z 517.462,A -85,B 0,C 180,E1 -4099.248,E2 -4099.248} C_VEL
LIN {X 0,Y 537.987,Z 517.466,A -85,B 0,C 180,E1 -4102.121,E2 -4102.121} C_VEL
LIN {X 0,Y 538.014,Z 517.465,A -85,B 0,C 180,E1 -4104.916,E2 -4104.916} C_VEL
LIN {X 0,Y 538.024,Z 517.468,A -85,B 0,C 180,E1 -4107.617,E2 -4107.617} C_VEL
LIN {X 0,Y 538.035,Z 517.46,A -85,B 0,C 180,E1 -4110.24,E2 -4110.24} C_VEL
LIN {X 0,Y 538.063,Z 517.456,A -85,B 0,C 180,E1 -4112.796,E2 -4112.796} C_VEL
LIN {X 0,Y 538.041,Z 517.467,A -85,B 0,C 180,E1 -4115.292,E2 -4115.292} C_VEL
LIN {X 0,Y 538.005,Z 517.465,A -85,B 0,C 180,E1 -4118.041,E2 -4118.041} C_VEL
LIN {X 0,Y 538.031,Z 517.46,A -85,B 0,C 180,E1 -4120.939,E2 -4120.939} C_VEL
LIN {X 0,Y 538.018,Z 517.47,A -85,B 0,C 180,E1 -4123.298,E2 -4123.298} C_VEL
LIN {X 0,Y 538.053,Z 517.464,A -85,B 0,C 180,E1 -4125.63,E2 -4125.63} C_VEL
LIN {X 0,Y 538.079,Z 517.453,A -85,B 0,C 180,E1 -4128.701,E2 -4128.701} C_VEL
LIN {X 0,Y 538.081,Z 517.458,A -85,B 0,C 180,E1 -4131.739,E2 -4131.739} C_VEL
LIN {X 0,Y 538.157,Z 517.446,A -85,B 0,C 180,E1 -4134.755,E2 -4134.755} C_VEL
LIN {X 0,Y 538.158,Z 517.448,A -85,B 0,C 180,E1 -4137.754,E2 -4137.754} C_VEL
LIN {X 0,Y 538.176,Z 517.444,A -85,B 0,C 180,E1 -4140.748,E2 -4140.748} C_VEL
LIN {X 0,Y 538.134,Z 517.451,A -85,B 0,C 180,E1 -4142.994,E2 -4142.994} C_VEL
LIN {X 0,Y 538.114,Z 517.452,A -85,B 0,C 180,E1 -4145.997,E2 -4145.997} C_VEL
LIN {X 0,Y 538.067,Z 517.46,A -85,B 0,C 180,E1 -4149.017,E2 -4149.017} C_VEL
LIN {X 0,Y 538.072,Z 517.457,A -85,B 0,C 180,E1 -4152.062,E2 -4152.062} C_VEL
LIN {X 0,Y 538.034,Z 517.467,A -85,B 0,C 180,E1 -4155.144,E2 -4155.144} C_VEL
LIN {X 0,Y 538.024,Z 517.462,A -85,B 0,C 180,E1 -4158.27,E2 -4158.27} C_VEL
LIN {X 0,Y 538.031,Z 517.462,A -85,B 0,C 180,E1 -4160.651,E2 -4160.651} C_VEL
LIN {X 0,Y 538.012,Z 517.467,A -85,B 0,C 180,E1 -4163.888,E2 -4163.888} C_VEL
LIN {X 0,Y 538.039,Z 517.461,A -85,B 0,C 180,E1 -4166.366,E2 -4166.366} C_VEL
LIN {X 0,Y 538.06,Z 517.466,A -85,B 0,C 180,E1 -4169.543,E2 -4169.543} C_VEL
LIN {X 0,Y 538.082,Z 517.655,A -85,B 0,C 180,E1 -4169.703,E2 -4169.703} C_VEL
LIN {X 0,Y 538.677,Z 522.106,A -85,B 0,C 180,E1 -4170.585,E2 -4170.585} C_VEL
LIN {X 0,Y 538.36,Z 536.663,A -85,B 0,C 180,E1 -4173.336,E2 -4173.336} C_VEL
LIN {X 0,Y 538.165,Z 547.187,A -85,B 0,C 180,E1 -4175.3,E2 -4175.3} C_VEL
LIN {X 0,Y 539.676,Z 557.478,A -85,B 0,C 180,E1 -4175.487,E2 -4175.487} C_VEL
LIN {X 0,Y 539.605,Z 575.669,A -85,B 0,C 180,E1 -4175.73,E2 -4175.73} C_VEL
LIN {X 0,Y 538.873,Z 581.511,A -85,B 0,C 180,E1 -4175.789,E2 -4175.789} C_VEL
LIN {X 0,Y 533.296,Z 600.517,A -85,B 0,C 180,E1 -4175.894,E2 -4175.894} C_VEL
LIN {X 0,Y 532.596,Z 606.358,A -85,B 0,C 180,E1 -4175.956,E2 -4175.956} C_VEL
LIN {X 0,Y 532.397,Z 654.894,A -85,B 0,C 180,E1 -4176.634,E2 -4176.634} C_VEL
LIN {X 0,Y 532.188,Z 668.502,A -85,B 0,C 180,E1 -4176.991,E2 -4176.991} C_VEL
LIN {X 0,Y 531.974,Z 681.254,A -85,B 0,C 180,E1 -4177.489,E2 -4177.489} C_VEL
LIN {X 0,Y 531.731,Z 694.1,A -85,B 0,C 180,E1 -4178.179,E2 -4178.179} C_VEL
LIN {X 0,Y 531.436,Z 705.037,A -85,B 0,C 180,E1 -4178.935,E2 -4178.935} C_VEL
LIN {X 0,Y 531.221,Z 715.976,A -85,B 0,C 180,E1 -4179.887,E2 -4179.887} C_VEL
LIN {X 0,Y 530.966,Z 725.126,A -85,B 0,C 180,E1 -4180.868,E2 -4180.868} C_VEL
LIN {X 0,Y 530.773,Z 733.386,A -85,B 0,C 180,E1 -4181.964,E2 -4181.964} C_VEL
LIN {X 0,Y 530.614,Z 741.13,A -85,B 0,C 180,E1 -4183.243,E2 -4183.243} C_VEL
LIN {X 0,Y 530.516,Z 747.42,A -85,B 0,C 180,E1 -4184.596,E2 -4184.596} C_VEL
LIN {X 0,Y 530.469,Z 751.296,A -85,B 0,C 180,E1 -4185.677,E2 -4185.677} C_VEL
LIN {X 0,Y 530.406,Z 754.291,A -85,B 0,C 180,E1 -4186.782,E2 -4186.782} C_VEL
LIN {X 0,Y 530.392,Z 756.403,A -85,B 0,C 180,E1 -4187.904,E2 -4187.904} C_VEL
LIN {X 0,Y 530.349,Z 757.643,A -85,B 0,C 180,E1 -4189.055,E2 -4189.055} C_VEL
LIN {X 0,Y 530.344,Z 757.913,A -85,B 0,C 180,E1 -4190.501,E2 -4190.501} C_VEL
LIN {X 0,Y 530.326,Z 757.272,A -85,B 0,C 180,E1 -4191.477,E2 -4191.477} C_VEL
LIN {X 0,Y 530.354,Z 755.612,A -85,B 0,C 180,E1 -4192.663,E2 -4192.663} C_VEL
LIN {X 0,Y 530.473,Z 752.759,A -85,B 0,C 180,E1 -4193.916,E2 -4193.916} C_VEL
LIN {X 0,Y 530.476,Z 748.315,A -85,B 0,C 180,E1 -4195.273,E2 -4195.273} C_VEL
LIN {X 0,Y 530.582,Z 742.583,A -85,B 0,C 180,E1 -4196.562,E2 -4196.562} C_VEL
LIN {X 0,Y 530.713,Z 735.687,A -85,B 0,C 180,E1 -4197.779,E2 -4197.779} C_VEL
LIN {X 0,Y 530.911,Z 727.566,A -85,B 0,C 180,E1 -4198.919,E2 -4198.919} C_VEL
LIN {X 0,Y 531.116,Z 717.725,A -85,B 0,C 180,E1 -4200.033,E2 -4200.033} C_VEL
LIN {X 0,Y 531.406,Z 707.26,A -85,B 0,C 180,E1 -4200.977,E2 -4200.977} C_VEL
LIN {X 0,Y 531.654,Z 696.21,A -85,B 0,C 180,E1 -4201.779,E2 -4201.779} C_VEL
LIN {X 0,Y 531.948,Z 684.2,A -85,B 0,C 180,E1 -4202.459,E2 -4202.459} C_VEL
LIN {X 0,Y 532.163,Z 671.355,A -85,B 0,C 180,E1 -4203.003,E2 -4203.003} C_VEL
LIN {X 0,Y 532.327,Z 659.055,A -85,B 0,C 180,E1 -4203.366,E2 -4203.366} C_VEL
LIN {X 0,Y 532.478,Z 643.521,A -85,B 0,C 180,E1 -4203.631,E2 -4203.631} C_VEL
LIN {X 0,Y 532.676,Z 556.007,A -85,B 0,C 180,E1 -4204.819,E2 -4204.819} C_VEL
LIN {X 0,Y 531.191,Z 547.406,A -85,B 0,C 180,E1 -4204.979,E2 -4204.979} C_VEL
LIN {X 0,Y 531.46,Z 532.683,A -85,B 0,C 180,E1 -4207.769,E2 -4207.769} C_VEL
LIN {X 0,Y 531.623,Z 521.981,A -85,B 0,C 180,E1 -4209.818,E2 -4209.818} C_VEL
LIN {X 0,Y 531.023,Z 518.342,A -85,B 0,C 180,E1 -4210.586,E2 -4210.586} C_VEL
LIN {X 0,Y 530.987,Z 518.344,A -85,B 0,C 180,E1 -4213.072,E2 -4213.072} C_VEL
LIN {X 0,Y 531.014,Z 518.336,A -85,B 0,C 180,E1 -4215.437,E2 -4215.437} C_VEL
LIN {X 0,Y 531.032,Z 518.337,A -85,B 0,C 180,E1 -4218.551,E2 -4218.551} C_VEL
LIN {X 0,Y 531.052,Z 518.329,A -85,B 0,C 180,E1 -4221.631,E2 -4221.631} C_VEL
LIN {X 0,Y 531.119,Z 518.327,A -85,B 0,C 180,E1 -4224.686,E2 -4224.686} C_VEL
LIN {X 0,Y 531.139,Z 518.318,A -85,B 0,C 180,E1 -4227.726,E2 -4227.726} C_VEL
LIN {X 0,Y 531.151,Z 518.324,A -85,B 0,C 180,E1 -4230.759,E2 -4230.759} C_VEL
LIN {X 0,Y 531.103,Z 518.331,A -85,B 0,C 180,E1 -4233.035,E2 -4233.035} C_VEL
LIN {X 0,Y 531.073,Z 518.326,A -85,B 0,C 180,E1 -4236.078,E2 -4236.078} C_VEL
LIN {X 0,Y 531.054,Z 518.33,A -85,B 0,C 180,E1 -4238.372,E2 -4238.372} C_VEL
LIN {X 0,Y 531.05,Z 518.331,A -85,B 0,C 180,E1 -4241.673,E2 -4241.673} C_VEL
LIN {X 0,Y 531.03,Z 518.34,A -85,B 0,C 180,E1 -4244.957,E2 -4244.957} C_VEL
LIN {X 0,Y 530.981,Z 518.339,A -85,B 0,C 180,E1 -4247.725,E2 -4247.725} C_VEL
LIN {X 0,Y 531.025,Z 518.332,A -85,B 0,C 180,E1 -4250.128,E2 -4250.128} C_VEL
LIN {X 0,Y 530.945,Z 518.344,A -85,B 0,C 180,E1 -4252.574,E2 -4252.574} C_VEL
LIN {X 0,Y 530.995,Z 518.344,A -85,B 0,C 180,E1 -4255.059,E2 -4255.059} C_VEL
LIN {X 0,Y 531.014,Z 518.337,A -85,B 0,C 180,E1 -4257.597,E2 -4257.597} C_VEL
LIN {X 0,Y 530.976,Z 518.34,A -85,B 0,C 180,E1 -4260.646,E2 -4260.646} C_VEL
LIN {X 0,Y 530.988,Z 518.339,A -85,B 0,C 180,E1 -4263.774,E2 -4263.774} C_VEL
LIN {X 0,Y 530.956,Z 518.342,A -85,B 0,C 180,E1 -4266.559,E2 -4266.559} C_VEL
LIN {X 0,Y 530.991,Z 518.344,A -85,B 0,C 180,E1 -4269.444,E2 -4269.444} C_VEL
LIN {X 0,Y 530.986,Z 518.337,A -85,B 0,C 180,E1 -4272.457,E2 -4272.457} C_VEL
LIN {X 0,Y 530.987,Z 518.343,A -85,B 0,C 180,E1 -4275.622,E2 -4275.622} C_VEL
LIN {X 0,Y 530.999,Z 518.336,A -85,B 0,C 180,E1 -4278.566,E2 -4278.566} C_VEL
LIN {X 0,Y 530.962,Z 518.349,A -85,B 0,C 180,E1 -4281.53,E2 -4281.53} C_VEL
LIN {X 0,Y 530.958,Z 518.341,A -85,B 0,C 180,E1 -4284.381,E2 -4284.381} C_VEL
LIN {X 0,Y 530.974,Z 518.343,A -85,B 0,C 180,E1 -4287.134,E2 -4287.134} C_VEL
LIN {X 0,Y 530.973,Z 518.344,A -85,B 0,C 180,E1 -4289.804,E2 -4289.804} C_VEL
LIN {X 0,Y 531.017,Z 518.333,A -85,B 0,C 180,E1 -4292.468,E2 -4292.468} C_VEL
LIN {X 0,Y 531.01,Z 518.336,A -85,B 0,C 180,E1 -4294.943,E2 -4294.943} C_VEL
LIN {X 0,Y 530.976,Z 518.34,A -85,B 0,C 180,E1 -4298.247,E2 -4298.247} C_VEL
LIN {X 0,Y 530.997,Z 518.336,A -85,B 0,C 180,E1 -4300.678,E2 -4300.678} C_VEL
LIN {X 0,Y 530.981,Z 518.34,A -85,B 0,C 180,E1 -4303.071,E2 -4303.071} C_VEL
LIN {X 0,Y 531.025,Z 518.338,A -85,B 0,C 180,E1 -4305.436,E2 -4305.436} C_VEL
LIN {X 0,Y 531.043,Z 518.33,A -85,B 0,C 180,E1 -4308.55,E2 -4308.55} C_VEL
LIN {X 0,Y 531.059,Z 518.336,A -85,B 0,C 180,E1 -4311.63,E2 -4311.63} C_VEL
LIN {X 0,Y 531.126,Z 518.32,A -85,B 0,C 180,E1 -4314.686,E2 -4314.686} C_VEL
LIN {X 0,Y 531.145,Z 518.326,A -85,B 0,C 180,E1 -4317.725,E2 -4317.725} C_VEL
LIN {X 0,Y 531.159,Z 518.316,A -85,B 0,C 180,E1 -4320.759,E2 -4320.759} C_VEL
LIN {X 0,Y 531.11,Z 518.322,A -85,B 0,C 180,E1 -4323.035,E2 -4323.035} C_VEL
LIN {X 0,Y 531.09,Z 518.331,A -85,B 0,C 180,E1 -4326.077,E2 -4326.077} C_VEL
LIN {X 0,Y 531.059,Z 518.331,A -85,B 0,C 180,E1 -4328.371,E2 -4328.371} C_VEL
LIN {X 0,Y 531.059,Z 518.333,A -85,B 0,C 180,E1 -4331.672,E2 -4331.672} C_VEL
LIN {X 0,Y 531.039,Z 518.331,A -85,B 0,C 180,E1 -4334.956,E2 -4334.956} C_VEL
LIN {X 0,Y 530.989,Z 518.342,A -85,B 0,C 180,E1 -4337.724,E2 -4337.724} C_VEL
LIN {X 0,Y 531.032,Z 518.34,A -85,B 0,C 180,E1 -4340.127,E2 -4340.127} C_VEL
LIN {X 0,Y 530.953,Z 518.344,A -85,B 0,C 180,E1 -4342.573,E2 -4342.573} C_VEL
LIN {X 0,Y 531.002,Z 518.335,A -85,B 0,C 180,E1 -4345.058,E2 -4345.058} C_VEL
LIN {X 0,Y 531.019,Z 518.335,A -85,B 0,C 180,E1 -4347.596,E2 -4347.596} C_VEL
LIN {X 0,Y 530.982,Z 518.34,A -85,B 0,C 180,E1 -4350.645,E2 -4350.645} C_VEL
LIN {X 0,Y 530.966,Z 518.343,A -85,B 0,C 180,E1 -4353.775,E2 -4353.775} C_VEL
LIN {X 0,Y 530.973,Z 518.343,A -85,B 0,C 180,E1 -4356.557,E2 -4356.557} C_VEL
LIN {X 0,Y 530.985,Z 518.341,A -85,B 0,C 180,E1 -4359.853,E2 -4359.853} C_VEL
LIN {X 0,Y 530.965,Z 518.346,A -85,B 0,C 180,E1 -4362.458,E2 -4362.458} C_VEL
LIN {X 0,Y 530.985,Z 518.338,A -85,B 0,C 180,E1 -4365.622,E2 -4365.622} C_VEL
LIN {X 0,Y 531.001,Z 518.341,A -85,B 0,C 180,E1 -4368.564,E2 -4368.564} C_VEL
LIN {X 0,Y 530.963,Z 518.34,A -85,B 0,C 180,E1 -4371.529,E2 -4371.529} C_VEL
LIN {X 0,Y 530.961,Z 518.35,A -85,B 0,C 180,E1 -4374.379,E2 -4374.379} C_VEL
LIN {X 0,Y 530.974,Z 518.339,A -85,B 0,C 180,E1 -4377.133,E2 -4377.133} C_VEL
LIN {X 0,Y 530.976,Z 518.341,A -85,B 0,C 180,E1 -4379.802,E2 -4379.802} C_VEL
LIN {X 0,Y 531.022,Z 518.342,A -85,B 0,C 180,E1 -4382.466,E2 -4382.466} C_VEL
LIN {X 0,Y 531.012,Z 518.342,A -85,B 0,C 180,E1 -4384.942,E2 -4384.942} C_VEL
LIN {X 0,Y 531.005,Z 518.464,A -85,B 0,C 180,E1 -4385.957,E2 -4385.957} C_VEL
LIN {X 0,Y 532.406,Z 526.227,A -85,B 0,C 180,E1 -4387.286,E2 -4387.286} C_VEL
LIN {X 0,Y 531.948,Z 545.321,A -85,B 0,C 180,E1 -4390.311,E2 -4390.311} C_VEL
LIN {X 0,Y 531.61,Z 561.852,A -85,B 0,C 180,E1 -4392.892,E2 -4392.892} C_VEL
LIN {X 0,Y 531.337,Z 575.773,A -85,B 0,C 180,E1 -4395.045,E2 -4395.045} C_VEL
LIN {X 0,Y 532.83,Z 585.967,A -85,B 0,C 180,E1 -4395.233,E2 -4395.233} C_VEL
LIN {X 0,Y 532.426,Z 683.836,A -85,B 0,C 180,E1 -4396.57,E2 -4396.57} C_VEL
LIN {X 0,Y 532.219,Z 697.157,A -85,B 0,C 180,E1 -4396.905,E2 -4396.905} C_VEL
LIN {X 0,Y 532.016,Z 709.345,A -85,B 0,C 180,E1 -4397.361,E2 -4397.361} C_VEL
LIN {X 0,Y 531.768,Z 721.236,A -85,B 0,C 180,E1 -4397.962,E2 -4397.962} C_VEL
LIN {X 0,Y 531.559,Z 733.179,A -85,B 0,C 180,E1 -4398.753,E2 -4398.753} C_VEL
LIN {X 0,Y 531.252,Z 743.593,A -85,B 0,C 180,E1 -4399.615,E2 -4399.615} C_VEL
LIN {X 0,Y 531.061,Z 752.104,A -85,B 0,C 180,E1 -4400.477,E2 -4400.477} C_VEL
LIN {X 0,Y 530.885,Z 759.953,A -85,B 0,C 180,E1 -4401.434,E2 -4401.434} C_VEL
LIN {X 0,Y 530.686,Z 767.615,A -85,B 0,C 180,E1 -4402.58,E2 -4402.58} C_VEL
LIN {X 0,Y 530.605,Z 774.674,A -85,B 0,C 180,E1 -4403.916,E2 -4403.916} C_VEL
LIN {X 0,Y 530.459,Z 779.369,A -85,B 0,C 180,E1 -4405.059,E2 -4405.059} C_VEL
LIN {X 0,Y 530.516,Z 782.955,A -85,B 0,C 180,E1 -4406.201,E2 -4406.201} C_VEL
LIN {X 0,Y 530.457,Z 784.805,A -85,B 0,C 180,E1 -4406.961,E2 -4406.961} C_VEL
LIN {X 0,Y 530.41,Z 786.192,A -85,B 0,C 180,E1 -4407.721,E2 -4407.721} C_VEL
LIN {X 0,Y 530.344,Z 787.785,A -85,B 0,C 180,E1 -4409.24,E2 -4409.24} C_VEL
LIN {X 0,Y 530.342,Z 788,A -85,B 0,C 180,E1 -4409.999,E2 -4409.999} C_VEL
LIN {X 0,Y 530.361,Z 787.185,A -85,B 0,C 180,E1 -4411.518,E2 -4411.518} C_VEL
LIN {X 0,Y 530.41,Z 786.198,A -85,B 0,C 180,E1 -4412.277,E2 -4412.277} C_VEL
LIN {X 0,Y 530.457,Z 784.812,A -85,B 0,C 180,E1 -4413.037,E2 -4413.037} C_VEL
LIN {X 0,Y 530.522,Z 781.898,A -85,B 0,C 180,E1 -4414.177,E2 -4414.177} C_VEL
LIN {X 0,Y 530.524,Z 777.952,A -85,B 0,C 180,E1 -4415.32,E2 -4415.32} C_VEL
LIN {X 0,Y 530.594,Z 772.288,A -85,B 0,C 180,E1 -4416.577,E2 -4416.577} C_VEL
LIN {X 0,Y 530.757,Z 765.243,A -85,B 0,C 180,E1 -4417.799,E2 -4417.799} C_VEL
LIN {X 0,Y 530.929,Z 757.001,A -85,B 0,C 180,E1 -4418.947,E2 -4418.947} C_VEL
LIN {X 0,Y 531.137,Z 748.551,A -85,B 0,C 180,E1 -4419.904,E2 -4419.904} C_VEL
LIN {X 0,Y 531.408,Z 738.105,A -85,B 0,C 180,E1 -4420.862,E2 -4420.862} C_VEL
LIN {X 0,Y 531.645,Z 727.153,A -85,B 0,C 180,E1 -4421.671,E2 -4421.671} C_VEL
LIN {X 0,Y 531.933,Z 716.425,A -85,B 0,C 180,E1 -4422.3,E2 -4422.3} C_VEL
LIN {X 0,Y 532.111,Z 704.789,A -85,B 0,C 180,E1 -4422.829,E2 -4422.829} C_VEL
LIN {X 0,Y 532.313,Z 691.341,A -85,B 0,C 180,E1 -4423.26,E2 -4423.26} C_VEL
LIN {X 0,Y 532.481,Z 678.072,A -85,B 0,C 180,E1 -4423.523,E2 -4423.523} C_VEL
LIN {X 0,Y 532.742,Z 584.257,A -85,B 0,C 180,E1 -4424.792,E2 -4424.792} C_VEL
LIN {X 0,Y 531.369,Z 575.728,A -85,B 0,C 180,E1 -4424.958,E2 -4424.958} C_VEL
LIN {X 0,Y 531.796,Z 554.096,A -85,B 0,C 180,E1 -4428.306,E2 -4428.306} C_VEL
LIN {X 0,Y 532.176,Z 535.067,A -85,B 0,C 180,E1 -4431.294,E2 -4431.294} C_VEL
LIN {X 0,Y 532.247,Z 524.85,A -85,B 0,C 180,E1 -4432.924,E2 -4432.924} C_VEL
LIN {X 0,Y 531.007,Z 518.342,A -85,B 0,C 180,E1 -4434.044,E2 -4434.044} C_VEL
LIN {X 0,Y 531.004,Z 518.339,A -85,B 0,C 180,E1 -4436.742,E2 -4436.742} C_VEL
LIN {X 0,Y 530.98,Z 518.348,A -85,B 0,C 180,E1 -4439.321,E2 -4439.321} C_VEL
LIN {X 0,Y 530.977,Z 518.342,A -85,B 0,C 180,E1 -4442.102,E2 -4442.102} C_VEL
LIN {X 0,Y 530.98,Z 518.341,A -85,B 0,C 180,E1 -4444.852,E2 -4444.852} C_VEL
LIN {X 0,Y 530.962,Z 518.351,A -85,B 0,C 180,E1 -4447.506,E2 -4447.506} C_VEL
LIN {X 0,Y 530.981,Z 518.34,A -85,B 0,C 180,E1 -4450.431,E2 -4450.431} C_VEL
LIN {X 0,Y 530.962,Z 518.352,A -85,B 0,C 180,E1 -4453.493,E2 -4453.493} C_VEL
LIN {X 0,Y 530.958,Z 518.343,A -85,B 0,C 180,E1 -4456.504,E2 -4456.504} C_VEL
LIN {X 0,Y 531.02,Z 518.341,A -85,B 0,C 180,E1 -4459.57,E2 -4459.57} C_VEL
LIN {X 0,Y 530.963,Z 518.34,A -85,B 0,C 180,E1 -4462.575,E2 -4462.575} C_VEL
LIN {X 0,Y 530.997,Z 518.344,A -85,B 0,C 180,E1 -4465.31,E2 -4465.31} C_VEL
LIN {X 0,Y 530.975,Z 518.341,A -85,B 0,C 180,E1 -4468.032,E2 -4468.032} C_VEL
LIN {X 0,Y 530.999,Z 518.338,A -85,B 0,C 180,E1 -4470.869,E2 -4470.869} C_VEL
LIN {X 0,Y 531.003,Z 518.341,A -85,B 0,C 180,E1 -4473.256,E2 -4473.256} C_VEL
LIN {X 0,Y 530.987,Z 518.338,A -85,B 0,C 180,E1 -4475.957,E2 -4475.957} C_VEL
LIN {X 0,Y 530.992,Z 518.341,A -85,B 0,C 180,E1 -4479.061,E2 -4479.061} C_VEL
LIN {X 0,Y 531.006,Z 518.336,A -85,B 0,C 180,E1 -4482.277,E2 -4482.277} C_VEL
LIN {X 0,Y 531.03,Z 518.341,A -85,B 0,C 180,E1 -4485.436,E2 -4485.436} C_VEL
LIN {X 0,Y 531.036,Z 518.33,A -85,B 0,C 180,E1 -4488.549,E2 -4488.549} C_VEL
LIN {X 0,Y 531.05,Z 518.335,A -85,B 0,C 180,E1 -4491.629,E2 -4491.629} C_VEL
LIN {X 0,Y 531.115,Z 518.322,A -85,B 0,C 180,E1 -4494.685,E2 -4494.685} C_VEL
LIN {X 0,Y 531.13,Z 518.324,A -85,B 0,C 180,E1 -4497.725,E2 -4497.725} C_VEL
LIN {X 0,Y 531.146,Z 518.32,A -85,B 0,C 180,E1 -4500.758,E2 -4500.758} C_VEL
LIN {X 0,Y 531.1,Z 518.327,A -85,B 0,C 180,E1 -4503.034,E2 -4503.034} C_VEL
LIN {X 0,Y 531.074,Z 518.329,A -85,B 0,C 180,E1 -4506.077,E2 -4506.077} C_VEL
LIN {X 0,Y 531.026,Z 518.339,A -85,B 0,C 180,E1 -4509.138,E2 -4509.138} C_VEL
LIN {X 0,Y 531.03,Z 518.334,A -85,B 0,C 180,E1 -4512.225,E2 -4512.225} C_VEL
LIN {X 0,Y 530.984,Z 518.348,A -85,B 0,C 180,E1 -4515.35,E2 -4515.35} C_VEL
LIN {X 0,Y 531.004,Z 518.341,A -85,B 0,C 180,E1 -4517.722,E2 -4517.722} C_VEL
LIN {X 0,Y 530.99,Z 518.341,A -85,B 0,C 180,E1 -4520.938,E2 -4520.938} C_VEL
LIN {X 0,Y 530.968,Z 518.342,A -85,B 0,C 180,E1 -4524.225,E2 -4524.225} C_VEL
LIN {X 0,Y 531.001,Z 518.34,A -85,B 0,C 180,E1 -4526.743,E2 -4526.743} C_VEL
LIN {X 0,Y 531.028,Z 518.454,A -85,B 0,C 180,E1 -4529.537,E2 -4529.537} C_VEL
LIN {X 0,Y 531.725,Z 523.035,A -85,B 0,C 180,E1 -4530.46,E2 -4530.46} C_VEL
LIN {X 0,Y 531.358,Z 539.262,A -85,B 0,C 180,E1 -4533.567,E2 -4533.567} C_VEL
LIN {X 0,Y 531.163,Z 547.46,A -85,B 0,C 180,E1 -4535.11,E2 -4535.11} C_VEL
LIN {X 0,Y 532.811,Z 558.224,A -85,B 0,C 180,E1 -4535.304,E2 -4535.304} C_VEL
LIN {X 0,Y 532.596,Z 606.358,A -85,B 0,C 180,E1 -4535.956,E2 -4535.956} C_VEL
LIN {X 0,Y 531.869,Z 612.204,A -85,B 0,C 180,E1 -4536.016,E2 -4536.016} C_VEL
LIN {X 0,Y 526.219,Z 631.198,A -85,B 0,C 180,E1 -4536.124,E2 -4536.124} C_VEL
LIN {X 0,Y 525.587,Z 637.04,A -85,B 0,C 180,E1 -4536.188,E2 -4536.188} C_VEL
LIN {X 0,Y 525.474,Z 656.845,A -85,B 0,C 180,E1 -4536.497,E2 -4536.497} C_VEL
LIN {X 0,Y 525.266,Z 669.54,A -85,B 0,C 180,E1 -4536.847,E2 -4536.847} C_VEL
LIN {X 0,Y 525.029,Z 681.771,A -85,B 0,C 180,E1 -4537.34,E2 -4537.34} C_VEL
LIN {X 0,Y 524.792,Z 694.347,A -85,B 0,C 180,E1 -4538.026,E2 -4538.026} C_VEL
LIN {X 0,Y 524.493,Z 704.869,A -85,B 0,C 180,E1 -4538.76,E2 -4538.76} C_VEL
LIN {X 0,Y 524.221,Z 715.383,A -85,B 0,C 180,E1 -4539.679,E2 -4539.679} C_VEL
LIN {X 0,Y 523.945,Z 725.027,A -85,B 0,C 180,E1 -4540.719,E2 -4540.719} C_VEL
LIN {X 0,Y 523.709,Z 733.898,A -85,B 0,C 180,E1 -4541.919,E2 -4541.919} C_VEL
LIN {X 0,Y 523.53,Z 741.467,A -85,B 0,C 180,E1 -4543.206,E2 -4543.206} C_VEL
LIN {X 0,Y 523.437,Z 746.475,A -85,B 0,C 180,E1 -4544.281,E2 -4544.281} C_VEL
LIN {X 0,Y 523.369,Z 751.589,A -85,B 0,C 180,E1 -4545.713,E2 -4545.713} C_VEL
LIN {X 0,Y 523.308,Z 754.367,A -85,B 0,C 180,E1 -4546.772,E2 -4546.772} C_VEL
LIN {X 0,Y 523.316,Z 756.325,A -85,B 0,C 180,E1 -4547.82,E2 -4547.82} C_VEL
LIN {X 0,Y 523.249,Z 757.518,A -85,B 0,C 180,E1 -4548.844,E2 -4548.844} C_VEL
LIN {X 0,Y 523.227,Z 757.989,A -85,B 0,C 180,E1 -4549.962,E2 -4549.962} C_VEL
LIN {X 0,Y 523.211,Z 757.566,A -85,B 0,C 180,E1 -4551.176,E2 -4551.176} C_VEL
LIN {X 0,Y 523.24,Z 756.114,A -85,B 0,C 180,E1 -4552.416,E2 -4552.416} C_VEL
LIN {X 0,Y 523.36,Z 753.248,A -85,B 0,C 180,E1 -4553.784,E2 -4553.784} C_VEL
LIN {X 0,Y 523.345,Z 749.555,A -85,B 0,C 180,E1 -4555.001,E2 -4555.001} C_VEL
LIN {X 0,Y 523.492,Z 744.123,A -85,B 0,C 180,E1 -4556.342,E2 -4556.342} C_VEL
LIN {X 0,Y 523.638,Z 737.882,A -85,B 0,C 180,E1 -4557.532,E2 -4557.532} C_VEL
LIN {X 0,Y 523.804,Z 730.663,A -85,B 0,C 180,E1 -4558.639,E2 -4558.639} C_VEL
LIN {X 0,Y 523.997,Z 723.196,A -85,B 0,C 180,E1 -4559.583,E2 -4559.583} C_VEL
LIN {X 0,Y 524.233,Z 713.199,A -85,B 0,C 180,E1 -4560.621,E2 -4560.621} C_VEL
LIN {X 0,Y 524.504,Z 702.749,A -85,B 0,C 180,E1 -4561.489,E2 -4561.489} C_VEL
LIN {X 0,Y 524.835,Z 690.951,A -85,B 0,C 180,E1 -4562.27,E2 -4562.27} C_VEL
LIN {X 0,Y 525.105,Z 678.889,A -85,B 0,C 180,E1 -4562.879,E2 -4562.879} C_VEL
LIN {X 0,Y 525.308,Z 665.758,A -85,B 0,C 180,E1 -4563.365,E2 -4563.365} C_VEL
LIN {X 0,Y 525.502,Z 653.342,A -85,B 0,C 180,E1 -4563.664,E2 -4563.664} C_VEL
LIN {X 0,Y 525.87,Z 557.157,A -85,B 0,C 180,E1 -4564.999,E2 -4564.999} C_VEL
LIN {X 0,Y 524.206,Z 547.461,A -85,B 0,C 180,E1 -4565.206,E2 -4565.206} C_VEL
LIN {X 0,Y 524.481,Z 533.102,A -85,B 0,C 180,E1 -4567.965,E2 -4567.965} C_VEL
LIN {X 0,Y 524.663,Z 523.686,A -85,B 0,C 180,E1 -4569.783,E2 -4569.783} C_VEL
LIN {X 0,Y 523.989,Z 519.218,A -85,B 0,C 180,E1 -4570.715,E2 -4570.715} C_VEL
LIN {X 0,Y 523.934,Z 519.219,A -85,B 0,C 180,E1 -4573.64,E2 -4573.64} C_VEL
LIN {X 0,Y 523.936,Z 519.218,A -85,B 0,C 180,E1 -4576.029,E2 -4576.029} C_VEL
LIN {X 0,Y 524.007,Z 519.21,A -85,B 0,C 180,E1 -4578.395,E2 -4578.395} C_VEL
LIN {X 0,Y 524,Z 519.208,A -85,B 0,C 180,E1 -4581.517,E2 -4581.517} C_VEL
LIN {X 0,Y 524.08,Z 519.203,A -85,B 0,C 180,E1 -4584.615,E2 -4584.615} C_VEL
LIN {X 0,Y 524.111,Z 519.194,A -85,B 0,C 180,E1 -4587.696,E2 -4587.696} C_VEL
LIN {X 0,Y 524.122,Z 519.199,A -85,B 0,C 180,E1 -4590.769,E2 -4590.769} C_VEL
LIN {X 0,Y 524.07,Z 519.207,A -85,B 0,C 180,E1 -4593.076,E2 -4593.076} C_VEL
LIN {X 0,Y 524.035,Z 519.203,A -85,B 0,C 180,E1 -4596.16,E2 -4596.16} C_VEL
LIN {X 0,Y 524.002,Z 519.21,A -85,B 0,C 180,E1 -4598.485,E2 -4598.485} C_VEL
LIN {X 0,Y 524.002,Z 519.208,A -85,B 0,C 180,E1 -4601.741,E2 -4601.741} C_VEL
LIN {X 0,Y 523.992,Z 519.218,A -85,B 0,C 180,E1 -4605.053,E2 -4605.053} C_VEL
LIN {X 0,Y 523.947,Z 519.214,A -85,B 0,C 180,E1 -4607.971,E2 -4607.971} C_VEL
LIN {X 0,Y 523.972,Z 519.212,A -85,B 0,C 180,E1 -4610.411,E2 -4610.411} C_VEL
LIN {X 0,Y 523.911,Z 519.224,A -85,B 0,C 180,E1 -4612.895,E2 -4612.895} C_VEL
LIN {X 0,Y 523.985,Z 519.21,A -85,B 0,C 180,E1 -4616.021,E2 -4616.021} C_VEL
LIN {X 0,Y 523.939,Z 519.219,A -85,B 0,C 180,E1 -4618.876,E2 -4618.876} C_VEL
LIN {X 0,Y 523.923,Z 519.222,A -85,B 0,C 180,E1 -4621.545,E2 -4621.545} C_VEL
LIN {X 0,Y 523.934,Z 519.216,A -85,B 0,C 180,E1 -4624.291,E2 -4624.291} C_VEL
LIN {X 0,Y 523.909,Z 519.226,A -85,B 0,C 180,E1 -4627.133,E2 -4627.133} C_VEL
LIN {X 0,Y 523.939,Z 519.215,A -85,B 0,C 180,E1 -4630.131,E2 -4630.131} C_VEL
LIN {X 0,Y 523.943,Z 519.215,A -85,B 0,C 180,E1 -4632.46,E2 -4632.46} C_VEL
LIN {X 0,Y 523.957,Z 519.222,A -85,B 0,C 180,E1 -4635.31,E2 -4635.31} C_VEL
LIN {X 0,Y 523.961,Z 519.213,A -85,B 0,C 180,E1 -4638.69,E2 -4638.69} C_VEL
LIN {X 0,Y 523.922,Z 519.221,A -85,B 0,C 180,E1 -4641.081,E2 -4641.081} C_VEL
LIN {X 0,Y 523.904,Z 519.224,A -85,B 0,C 180,E1 -4643.826,E2 -4643.826} C_VEL
LIN {X 0,Y 523.946,Z 519.214,A -85,B 0,C 180,E1 -4646.636,E2 -4646.636} C_VEL
LIN {X 0,Y 523.96,Z 519.22,A -85,B 0,C 180,E1 -4649.356,E2 -4649.356} C_VEL
LIN {X 0,Y 523.981,Z 519.211,A -85,B 0,C 180,E1 -4652.282,E2 -4652.282} C_VEL
LIN {X 0,Y 523.957,Z 519.213,A -85,B 0,C 180,E1 -4654.582,E2 -4654.582} C_VEL
LIN {X 0,Y 523.915,Z 519.221,A -85,B 0,C 180,E1 -4657.107,E2 -4657.107} C_VEL
LIN {X 0,Y 523.984,Z 519.215,A -85,B 0,C 180,E1 -4659.867,E2 -4659.867} C_VEL
LIN {X 0,Y 523.963,Z 519.212,A -85,B 0,C 180,E1 -4662.838,E2 -4662.838} C_VEL
LIN {X 0,Y 523.983,Z 519.213,A -85,B 0,C 180,E1 -4665.236,E2 -4665.236} C_VEL
LIN {X 0,Y 524.019,Z 519.206,A -85,B 0,C 180,E1 -4668.395,E2 -4668.395} C_VEL
LIN {X 0,Y 524.007,Z 519.213,A -85,B 0,C 180,E1 -4671.516,E2 -4671.516} C_VEL
LIN {X 0,Y 524.087,Z 519.197,A -85,B 0,C 180,E1 -4674.614,E2 -4674.614} C_VEL
LIN {X 0,Y 524.117,Z 519.201,A -85,B 0,C 180,E1 -4677.695,E2 -4677.695} C_VEL
LIN {X 0,Y 524.129,Z 519.191,A -85,B 0,C 180,E1 -4680.769,E2 -4680.769} C_VEL
LIN {X 0,Y 524.077,Z 519.198,A -85,B 0,C 180,E1 -4683.075,E2 -4683.075} C_VEL
LIN {X 0,Y 524.053,Z 519.206,A -85,B 0,C 180,E1 -4686.159,E2 -4686.159} C_VEL
LIN {X 0,Y 524.007,Z 519.208,A -85,B 0,C 180,E1 -4688.484,E2 -4688.484} C_VEL
LIN {X 0,Y 524.01,Z 519.213,A -85,B 0,C 180,E1 -4691.739,E2 -4691.739} C_VEL
LIN {X 0,Y 524.001,Z 519.207,A -85,B 0,C 180,E1 -4695.052,E2 -4695.052} C_VEL
LIN {X 0,Y 523.955,Z 519.222,A -85,B 0,C 180,E1 -4697.97,E2 -4697.97} C_VEL
LIN {X 0,Y 523.979,Z 519.214,A -85,B 0,C 180,E1 -4700.41,E2 -4700.41} C_VEL
LIN {X 0,Y 523.918,Z 519.218,A -85,B 0,C 180,E1 -4702.894,E2 -4702.894} C_VEL
LIN {X 0,Y 523.991,Z 519.217,A -85,B 0,C 180,E1 -4706.02,E2 -4706.02} C_VEL
LIN {X 0,Y 523.943,Z 519.215,A -85,B 0,C 180,E1 -4708.875,E2 -4708.875} C_VEL
LIN {X 0,Y 523.928,Z 519.218,A -85,B 0,C 180,E1 -4711.544,E2 -4711.544} C_VEL
LIN {X 0,Y 523.932,Z 519.224,A -85,B 0,C 180,E1 -4714.291,E2 -4714.291} C_VEL
LIN {X 0,Y 523.918,Z 519.218,A -85,B 0,C 180,E1 -4717.132,E2 -4717.132} C_VEL
LIN {X 0,Y 523.945,Z 519.222,A -85,B 0,C 180,E1 -4720.13,E2 -4720.13} C_VEL
LIN {X 0,Y 523.925,Z 519.223,A -85,B 0,C 180,E1 -4722.456,E2 -4722.456} C_VEL
LIN {X 0,Y 523.949,Z 519.214,A -85,B 0,C 180,E1 -4725.31,E2 -4725.31} C_VEL
LIN {X 0,Y 523.963,Z 519.216,A -85,B 0,C 180,E1 -4728.689,E2 -4728.689} C_VEL
LIN {X 0,Y 523.924,Z 519.218,A -85,B 0,C 180,E1 -4731.08,E2 -4731.08} C_VEL
LIN {X 0,Y 523.907,Z 519.221,A -85,B 0,C 180,E1 -4733.825,E2 -4733.825} C_VEL
LIN {X 0,Y 523.948,Z 519.22,A -85,B 0,C 180,E1 -4736.635,E2 -4736.635} C_VEL
LIN {X 0,Y 523.963,Z 519.214,A -85,B 0,C 180,E1 -4739.355,E2 -4739.355} C_VEL
LIN {X 0,Y 523.985,Z 519.217,A -85,B 0,C 180,E1 -4742.281,E2 -4742.281} C_VEL
LIN {X 0,Y 523.959,Z 519.222,A -85,B 0,C 180,E1 -4744.581,E2 -4744.581} C_VEL
LIN {X 0,Y 523.984,Z 519.399,A -85,B 0,C 180,E1 -4745.792,E2 -4745.792} C_VEL
LIN {X 0,Y 525.45,Z 527.359,A -85,B 0,C 180,E1 -4747.176,E2 -4747.176} C_VEL
LIN {X 0,Y 525.008,Z 545.159,A -85,B 0,C 180,E1 -4750.04,E2 -4750.04} C_VEL
LIN {X 0,Y 524.616,Z 561.691,A -85,B 0,C 180,E1 -4752.657,E2 -4752.657} C_VEL
LIN {X 0,Y 524.317,Z 575.65,A -85,B 0,C 180,E1 -4754.847,E2 -4754.847} C_VEL
LIN {X 0,Y 525.979,Z 586.938,A -85,B 0,C 180,E1 -4755.054,E2 -4755.054} C_VEL
LIN {X 0,Y 525.528,Z 683.454,A -85,B 0,C 180,E1 -4756.391,E2 -4756.391} C_VEL
LIN {X 0,Y 525.294,Z 696.837,A -85,B 0,C 180,E1 -4756.729,E2 -4756.729} C_VEL
LIN {X 0,Y 525.07,Z 710.189,A -85,B 0,C 180,E1 -4757.24,E2 -4757.24} C_VEL
LIN {X 0,Y 524.782,Z 721.993,A -85,B 0,C 180,E1 -4757.86,E2 -4757.86} C_VEL
LIN {X 0,Y 524.52,Z 734.309,A -85,B 0,C 180,E1 -4758.698,E2 -4758.698} C_VEL
LIN {X 0,Y 524.215,Z 744.524,A -85,B 0,C 180,E1 -4759.572,E2 -4759.572} C_VEL
LIN {X 0,Y 523.977,Z 753.712,A -85,B 0,C 180,E1 -4760.542,E2 -4760.542} C_VEL
LIN {X 0,Y 523.76,Z 762.662,A -85,B 0,C 180,E1 -4761.705,E2 -4761.705} C_VEL
LIN {X 0,Y 523.585,Z 769.842,A -85,B 0,C 180,E1 -4762.867,E2 -4762.867} C_VEL
LIN {X 0,Y 523.544,Z 776.362,A -85,B 0,C 180,E1 -4764.221,E2 -4764.221} C_VEL
LIN {X 0,Y 523.361,Z 780.673,A -85,B 0,C 180,E1 -4765.378,E2 -4765.378} C_VEL
LIN {X 0,Y 523.444,Z 782.955,A -85,B 0,C 180,E1 -4766.15,E2 -4766.15} C_VEL
LIN {X 0,Y 523.368,Z 784.804,A -85,B 0,C 180,E1 -4766.92,E2 -4766.92} C_VEL
LIN {X 0,Y 523.334,Z 786.191,A -85,B 0,C 180,E1 -4767.69,E2 -4767.69} C_VEL
LIN {X 0,Y 523.25,Z 787.784,A -85,B 0,C 180,E1 -4769.229,E2 -4769.229} C_VEL
LIN {X 0,Y 523.246,Z 788,A -85,B 0,C 180,E1 -4769.999,E2 -4769.999} C_VEL
LIN {X 0,Y 523.274,Z 787.184,A -85,B 0,C 180,E1 -4771.538,E2 -4771.538} C_VEL
LIN {X 0,Y 523.334,Z 786.197,A -85,B 0,C 180,E1 -4772.308,E2 -4772.308} C_VEL
LIN {X 0,Y 523.367,Z 784.812,A -85,B 0,C 180,E1 -4773.078,E2 -4773.078} C_VEL
LIN {X 0,Y 523.441,Z 781.898,A -85,B 0,C 180,E1 -4774.234,E2 -4774.234} C_VEL
LIN {X 0,Y 523.464,Z 777.952,A -85,B 0,C 180,E1 -4775.392,E2 -4775.392} C_VEL
LIN {X 0,Y 523.519,Z 772.752,A -85,B 0,C 180,E1 -4776.576,E2 -4776.576} C_VEL
LIN {X 0,Y 523.664,Z 766.472,A -85,B 0,C 180,E1 -4777.712,E2 -4777.712} C_VEL
LIN {X 0,Y 523.853,Z 758.443,A -85,B 0,C 180,E1 -4778.874,E2 -4778.874} C_VEL
LIN {X 0,Y 524.077,Z 750.255,A -85,B 0,C 180,E1 -4779.844,E2 -4779.844} C_VEL
LIN {X 0,Y 524.35,Z 740.268,A -85,B 0,C 180,E1 -4780.814,E2 -4780.814} C_VEL
LIN {X 0,Y 524.639,Z 728.897,A -85,B 0,C 180,E1 -4781.695,E2 -4781.695} C_VEL
LIN {X 0,Y 524.922,Z 717.932,A -85,B 0,C 180,E1 -4782.368,E2 -4782.368} C_VEL
LIN {X 0,Y 525.157,Z 705.675,A -85,B 0,C 180,E1 -4782.952,E2 -4782.952} C_VEL
LIN {X 0,Y 525.364,Z 692.79,A -85,B 0,C 180,E1 -4783.39,E2 -4783.39} C_VEL
LIN {X 0,Y 525.575,Z 679.103,A -85,B 0,C 180,E1 -4783.68,E2 -4783.68} C_VEL
LIN {X 0,Y 525.869,Z 585.086,A -85,B 0,C 180,E1 -4784.972,E2 -4784.972} C_VEL
LIN {X 0,Y 524.333,Z 575.534,A -85,B 0,C 180,E1 -4785.159,E2 -4785.159} C_VEL
LIN {X 0,Y 524.813,Z 554.118,A -85,B 0,C 180,E1 -4788.523,E2 -4788.523} C_VEL
LIN {X 0,Y 525.218,Z 534.864,A -85,B 0,C 180,E1 -4791.59,E2 -4791.59} C_VEL
LIN {X 0,Y 525.413,Z 527.221,A -85,B 0,C 180,E1 -4792.823,E2 -4792.823} C_VEL
LIN {X 0,Y 523.956,Z 519.22,A -85,B 0,C 180,E1 -4794.23,E2 -4794.23} C_VEL
LIN {X 0,Y 523.952,Z 519.221,A -85,B 0,C 180,E1 -4797.131,E2 -4797.131} C_VEL
LIN {X 0,Y 523.94,Z 519.224,A -85,B 0,C 180,E1 -4799.755,E2 -4799.755} C_VEL
LIN {X 0,Y 523.937,Z 519.217,A -85,B 0,C 180,E1 -4802.448,E2 -4802.448} C_VEL
LIN {X 0,Y 523.928,Z 519.223,A -85,B 0,C 180,E1 -4805.224,E2 -4805.224} C_VEL
LIN {X 0,Y 523.913,Z 519.222,A -85,B 0,C 180,E1 -4808.1,E2 -4808.1} C_VEL
LIN {X 0,Y 523.94,Z 519.221,A -85,B 0,C 180,E1 -4811.09,E2 -4811.09} C_VEL
LIN {X 0,Y 523.936,Z 519.218,A -85,B 0,C 180,E1 -4814.226,E2 -4814.226} C_VEL
LIN {X 0,Y 523.915,Z 519.221,A -85,B 0,C 180,E1 -4816.832,E2 -4816.832} C_VEL
LIN {X 0,Y 523.971,Z 519.214,A -85,B 0,C 180,E1 -4819.922,E2 -4819.922} C_VEL
LIN {X 0,Y 523.906,Z 519.221,A -85,B 0,C 180,E1 -4822.867,E2 -4822.867} C_VEL
LIN {X 0,Y 523.939,Z 519.221,A -85,B 0,C 180,E1 -4825.71,E2 -4825.71} C_VEL
LIN {X 0,Y 523.925,Z 519.217,A -85,B 0,C 180,E1 -4828.456,E2 -4828.456} C_VEL
LIN {X 0,Y 523.943,Z 519.22,A -85,B 0,C 180,E1 -4831.125,E2 -4831.125} C_VEL
LIN {X 0,Y 523.977,Z 519.213,A -85,B 0,C 180,E1 -4833.979,E2 -4833.979} C_VEL
LIN {X 0,Y 523.927,Z 519.215,A -85,B 0,C 180,E1 -4836.27,E2 -4836.27} C_VEL
LIN {X 0,Y 523.938,Z 519.217,A -85,B 0,C 180,E1 -4838.766,E2 -4838.766} C_VEL
LIN {X 0,Y 523.945,Z 519.219,A -85,B 0,C 180,E1 -4841.22,E2 -4841.22} C_VEL
LIN {X 0,Y 523.931,Z 519.221,A -85,B 0,C 180,E1 -4843.638,E2 -4843.638} C_VEL
LIN {X 0,Y 523.935,Z 519.218,A -85,B 0,C 180,E1 -4846.028,E2 -4846.028} C_VEL
LIN {X 0,Y 524.001,Z 519.206,A -85,B 0,C 180,E1 -4848.393,E2 -4848.393} C_VEL
LIN {X 0,Y 523.998,Z 519.215,A -85,B 0,C 180,E1 -4851.516,E2 -4851.516} C_VEL
LIN {X 0,Y 524.076,Z 519.199,A -85,B 0,C 180,E1 -4854.613,E2 -4854.613} C_VEL
LIN {X 0,Y 524.102,Z 519.2,A -85,B 0,C 180,E1 -4857.694,E2 -4857.694} C_VEL
LIN {X 0,Y 524.115,Z 519.195,A -85,B 0,C 180,E1 -4860.768,E2 -4860.768} C_VEL
LIN {X 0,Y 524.067,Z 519.204,A -85,B 0,C 180,E1 -4863.075,E2 -4863.075} C_VEL
LIN {X 0,Y 524.035,Z 519.205,A -85,B 0,C 180,E1 -4866.159,E2 -4866.159} C_VEL
LIN {X 0,Y 523.993,Z 519.217,A -85,B 0,C 180,E1 -4869.262,E2 -4869.262} C_VEL
LIN {X 0,Y 524.012,Z 519.212,A -85,B 0,C 180,E1 -4871.751,E2 -4871.751} C_VEL
LIN {X 0,Y 523.98,Z 519.216,A -85,B 0,C 180,E1 -4875.052,E2 -4875.052} C_VEL
LIN {X 0,Y 523.952,Z 519.217,A -85,B 0,C 180,E1 -4877.969,E2 -4877.969} C_VEL
